(* Monitoring Prisma *)
	IF (T_Visu.T_PlcParam.dwActualPage = 430) THEN
		FailingEdgePrisma(CLK:=TRUE);
		RisingEdgePrisma(CLK:=(T_Visu.T_PlcParam.dwActualPage = 430));
		IF RisingEdgePrisma.Q THEN
		(* 0= 3 value prisma, 1 = 3 value prisma input para, 2 = 2 value prisma, 3 = 2 value prisma input para *)
			IF (T_Visu.ptrT_ExchgParam^.T_StationCommon.T_PrismPara.bStateInputPrisma = 1) THEN
				T_Visu.ptrT_ExchgParam^.T_StationCommon.T_PrismPara.bStateInputPrisma:=0;
			END_IF;
			IF (T_Visu.ptrT_ExchgParam^.T_StationCommon.T_PrismPara.bStateInputPrisma = 3) THEN
				T_Visu.ptrT_ExchgParam^.T_StationCommon.T_PrismPara.bStateInputPrisma:=2;
			END_IF;
		END_IF;
	ELSE
		RisingEdgePrisma(CLK:=FALSE);
		FailingEdgePrisma(CLK:=FALSE);
		(*If the page changes, then copy again the settled value *)
		IF FailingEdgePrisma.Q THEN
			T_Visu.ptrT_ExchgParam^.T_StationCommon.T_PrismPara:=T_NovRAM.T_Data.T_ProcessImageData.T_PrismPara;
		END_IF;
	END_IF

(* Tmp timer *)
	TimerONTmp(IN:=TRUE);



(************************************************************************************************************************************************************************)
(***************                                          start of the management for call a function of the visualisation interface                                           ********************)
(************************************************************************************************************************************************************************)
CtrlVisuFunction;
(************************************************************************************************************************************************************************)
(***************                                          end of the management for call a function of the visualisation interface                                           ********************)
(************************************************************************************************************************************************************************)



(************************************************************************************************************************************************************************)
(***************                                                   start of the checking of the activation of an visualisation action                                                   ********************)
(************************************************************************************************************************************************************************)
(* check if Action is Acitve and if the power supply is on, otherwise block the action *)
	xTmp:=	xStopAxis OR xMoveRelPosition OR xMoveAbsPosition OR xMoveContinousVel OR xSwitchMasterSlave OR xToggleAxisPower OR xResetAxis OR xReferenceAxis OR xTeachPosition OR xCylBrake;
	xTmp:=	xTmp OR xToggleCylinderState OR xToolTensForceAdd OR xToolTensForceAddMore OR xToolTensForceSub OR xToolTensForceSubMore;
	xTmp:=	xTmp OR xToolFeederMoveStartPos OR xToggleAllAxisPower OR xCalcAngleRefIndex OR xToolFeederMoveLoadPos;
	xTmp:=	xTmp OR xActivateStationFunction OR xActionProcStation OR xActionProcMachine OR xStopProcess;
	xTmp:=	xTmp OR xOverlayGrindFeedSetPlung OR xOverlayMeasureToolDia OR xFctCorrectionToolDiameter OR xAction_LoadProfileToProcessImage;
	xTmp:=	xTmp OR ((T_Visu.T_PlcParam.dwActualPage = 430) AND xAction_SaveNovRAM);
(*SOA 31.01.2023  { *)
	xTmp:= xTmp OR (T_Visu.T_PlcParam.dwActualPage = 141) ;
(*SOA 31.01.2023  } *)
	IF xTmp THEN
		IF NOT(T_TwinSafeOut.QxContactor_K3) OR NOT(T_TwinSafeOut.QxContactor_K4) THEN
			xStopAxis:=xMoveRelPosition:=xMoveAbsPosition:=xMoveContinousVel:=xSwitchMasterSlave:=xToggleAxisPower:=xResetAxis:=xReferenceAxis:=xTeachPosition:=xCylBrake:=FALSE;
			xToggleCylinderState:=xToolTensForceAdd:=xToolTensForceAddMore:=xToolTensForceSub:=xToolTensForceSubMore:=FALSE;
			xToolFeederMoveStartPos:=xToggleAllAxisPower:=xCalcAngleRefIndex:=xToolFeederMoveLoadPos:= FALSE;
			xActivateStationFunction:=xActionProcStation:=xActionProcMachine:=xStopProcess:=FALSE;
			xOverlayGrindFeedSetPlung:=xOverlayMeasureToolDia:=xFctCorrectionToolDiameter:=xAction_LoadProfileToProcessImage:=FALSE;
			T_Visu.ptrT_ExchgParam^.T_FunctionCommon.xOpenOverlayMessageBox:=FALSE;
			T_Visu.ptrT_ExchgParam^.T_FunctionCommon.xOpenOverlayMeasureInput:=FALSE;
			T_Visu.ptrT_ExchgParam^.T_FunctionCommon.xOpenOverlaySetGrindPlunge:=FALSE;
			T_Visu.ptrT_ExchgParam^.T_FunctionCommon.xSaveButton:=FALSE;
			T_Visu.ptrT_ExchgParam^.T_FunctionCommon.xExitButton:=FALSE;
			T_Visu.ptrT_ExchgParam^.T_FunctionCommon.xHideProgressbar:=FALSE;
			xAction_SaveNovRAM:=FALSE;
			T_Visu.T_CtrleAction.xDone:=TRUE;
			T_Visu.T_CtrleAction.xNotReady:=FALSE;
			T_Visu.T_CtrleAction.xErr:=FALSE;
			T_Visu.T_CtrleAction.udiErrorID:=0;
			tTimeOutAction:=T#0s;
			TimerAction(IN:=FALSE);
			(* Display Message --> Switch first the energy supply ON *)
			T_ExchgParam.T_Visu.T_Message.iState:=120;
			xBlockConfirmMessage:=TRUE;
			TONTimeWaitMsg(IN:=FALSE);
		END_IF;
	END_IF;
	IF (T_ExchgParam.T_Visu.T_Message.iState = 120) THEN
		TONTimeWaitMsg(IN:=TRUE,PT:=T#3s);
		IF TONTimeWaitMsg.Q THEN
			T_ExchgParam.T_Visu.T_Message.iState:=0;	(* Deactivate again the message *)
		END_IF;
	ELSE
		TONTimeWaitMsg(IN:=FALSE);
	END_IF;

(* check if an error is active, otherwise block the action *)
	IF (T_ExchgParam.T_Visu.T_Message.iState = 401) THEN
		xTmp:=	xStopAxis OR xMoveRelPosition OR xMoveAbsPosition OR xMoveContinousVel OR xSwitchMasterSlave OR xToggleAxisPower OR xResetAxis OR xReferenceAxis OR xTeachPosition OR xCylBrake;
		xTmp:=	xTmp OR xToggleCylinderState OR xToolTensForceAdd OR xToolTensForceAddMore OR xToolTensForceSub OR xToolTensForceSubMore;
		xTmp:=	xTmp OR xToolFeederMoveStartPos OR xToggleAllAxisPower OR xCalcAngleRefIndex OR xToolFeederMoveLoadPos;
		xTmp:=	xTmp OR xActivateStationFunction OR xActionProcStation OR xActionProcMachine OR xStopProcess;
		xTmp:=	xTmp OR xOverlayGrindFeedSetPlung OR xOverlayMeasureToolDia OR xFctCorrectionToolDiameter OR xAction_LoadProfileToProcessImage;
		xTmp:=	xTmp OR ((T_Visu.T_PlcParam.dwActualPage = 430) AND xAction_SaveNovRAM);
		IF xTmp THEN
			xStopAxis:=xMoveRelPosition:=xMoveAbsPosition:=xMoveContinousVel:=xSwitchMasterSlave:=xToggleAxisPower:=xResetAxis:=xReferenceAxis:=xTeachPosition:=xCylBrake:=FALSE;
			xToggleCylinderState:=xToolTensForceAdd:=xToolTensForceAddMore:=xToolTensForceSub:=xToolTensForceSubMore:=FALSE;
			xToolFeederMoveStartPos:=xToggleAllAxisPower:=xCalcAngleRefIndex:=xToolFeederMoveLoadPos:=FALSE;
			xActivateStationFunction:=xActionProcStation:=xActionProcMachine:=xStopProcess:=FALSE;
			xOverlayGrindFeedSetPlung:=xOverlayMeasureToolDia:=xFctCorrectionToolDiameter:=xAction_LoadProfileToProcessImage:=FALSE;
			xAction_SaveNovRAM:=FALSE;
			T_Visu.T_CtrleAction.xDone:=TRUE;
			T_Visu.T_CtrleAction.xNotReady:=FALSE;
			T_Visu.T_CtrleAction.xErr:=FALSE;
			T_Visu.T_CtrleAction.udiErrorID:=0;
			tTimeOutAction:=T#0s;
			TimerAction(IN:=FALSE);
		END_IF;
	END_IF;
(************************************************************************************************************************************************************************)
(***************                                                   end of the checking of the activation of an visualisation action                                                   ********************)
(************************************************************************************************************************************************************************)

(************************************************************************************************************************************************************************)
(***************                                             start for the section for defined function of the visualisation interface                                               ********************)
(************************************************************************************************************************************************************************)
VisuFunction_SetParameterPage;

(* Action change page from navigation panel *)
	IF xNavPanelChangePage OR xBtPanelLeftChangePage OR  xBtPanelRightChangePage OR xNextPageVertical THEN
		(* Step change page from navigation panel *)
		CASE iStepAction OF
		(* check visu *)
		1:	xTmp:=	T_Visu.T_CtrleVisu.xDone
					AND NOT(T_Visu.T_CtrleVisu.xExecute)
					AND NOT(T_Visu.T_CtrleVisu.xErr);
			IF xTmp THEN
				(* next Step *)
				iStepAction :=10;
				xStepActionDone:=FALSE;
			(* activ error *)
			ELSE iStepAction:=95; END_IF
		(* activ change page *)
		10:	T_Visu.T_CtrleVisu.xExecute:=TRUE;
			T_Visu.T_CtrleVisu.iFunction:=1;
			T_Visu.ptrT_ExchgParam^.T_Config.iEditParam:=0;
			IF xNavPanelChangePage THEN
				T_Visu.T_PlcParam.dwSetNewPage:=INT_TO_DWORD(T_Visu.T_CtrleAction.iFunction - 10000);
				CASE T_Visu.ptrT_ExchgParam^.T_Visu.bActivSpecialLayer OF
					0:	IF awNormalLayerActivPage[wTmpNormalLayerActivTask] <> 0 AND awNormalLayerActivPage[wTmpNormalLayerActivTask] <> T_Visu.T_PlcParam.dwSetNewPage THEN
							T_Visu.T_PlcParam.dwSetNewPage:=awNormalLayerActivPage[wTmpNormalLayerActivTask];
						END_IF;
					1:	IF awSpecialLayerGeneralActivPage[wTmpSpecialLayerGeneralActivTask] <> 0 AND awSpecialLayerGeneralActivPage[wTmpSpecialLayerGeneralActivTask] <> T_Visu.T_PlcParam.dwSetNewPage THEN
							T_Visu.T_PlcParam.dwSetNewPage:=awSpecialLayerGeneralActivPage[wTmpSpecialLayerGeneralActivTask];
						END_IF;
					2:	IF awSpecialLayerToolRotActivPage[wTmpSpecialLayerToolRotActivTask] <> 0 AND awSpecialLayerToolRotActivPage[wTmpSpecialLayerToolRotActivTask] <> T_Visu.T_PlcParam.dwSetNewPage THEN
							T_Visu.T_PlcParam.dwSetNewPage:=awSpecialLayerToolRotActivPage[wTmpSpecialLayerToolRotActivTask];
						END_IF;
					3:	IF awSpecialLayerWireFeedActivPage[wTmpSpecialLayerWireFeedActivTask] <> 0 AND awSpecialLayerWireFeedActivPage[wTmpSpecialLayerWireFeedActivTask] <> T_Visu.T_PlcParam.dwSetNewPage THEN
							T_Visu.T_PlcParam.dwSetNewPage:=awSpecialLayerWireFeedActivPage[wTmpSpecialLayerWireFeedActivTask];
						END_IF;
					4:	IF awSpecialLayerGrindAxisActivPage[wTmpSpecialLayerGrindAxisActivTask] <> 0 AND awSpecialLayerGrindAxisActivPage[wTmpSpecialLayerGrindAxisActivTask] <> T_Visu.T_PlcParam.dwSetNewPage THEN
							T_Visu.T_PlcParam.dwSetNewPage:=awSpecialLayerGrindAxisActivPage[wTmpSpecialLayerGrindAxisActivTask];
						END_IF;
				END_CASE;
			END_IF;
			IF xBtPanelLeftChangePage THEN
				T_Visu.T_PlcParam.dwSetNewPage:=dwSetNewPage;
				T_Visu.ptrT_ExchgParam^.T_Config.xBlockParaListNavi:=FALSE;
				T_Visu.ptrT_ExchgParam^.T_Config.xBlockParaListNavi1:=TRUE;
				T_Visu.ptrT_ExchgParam^.T_Config.xBlockProfilList:=TRUE;
			END_IF;
(*SOA*)
			IF xBtPanelRightChangePage THEN
				T_Visu.T_PlcParam.dwSetNewPage:=dwSetNewPage;
				T_Visu.ptrT_ExchgParam^.T_Config.xBlockParaListNavi:=FALSE;
				T_Visu.ptrT_ExchgParam^.T_Config.xBlockParaListNavi1:=TRUE;
				T_Visu.ptrT_ExchgParam^.T_Config.xBlockProfilList:=TRUE;
			END_IF;
(*SOA*)
			IF xNextPageVertical THEN
				IF (T_Visu.T_PageIndex[T_Visu.T_PlcParam.dwActualPage + 1].iIndexConfigPage <> 0) THEN
					T_Visu.T_PlcParam.dwSetNewPage:=T_Visu.T_PlcParam.dwActualPage + 1;
				ELSE
					FOR ii:=1 TO 9 DO
						IF (T_Visu.T_PageIndex[T_Visu.T_PlcParam.dwActualPage - 1].iIndexConfigPage <> 0) THEN
							T_Visu.T_PlcParam.dwActualPage:=T_Visu.T_PlcParam.dwActualPage - 1;
						ELSE
							T_Visu.T_PlcParam.dwSetNewPage:=T_Visu.T_PlcParam.dwActualPage;
							EXIT;
						END_IF;
					END_FOR;
				END_IF;
				CASE T_Visu.ptrT_ExchgParam^.T_Visu.bActivSpecialLayer OF
					0:	awNormalLayerActivPage[wTmpNormalLayerActivTask]:=DWORD_TO_WORD(T_Visu.T_PlcParam.dwSetNewPage);
					1:	awSpecialLayerGeneralActivPage[wTmpSpecialLayerGeneralActivTask]:=DWORD_TO_WORD(T_Visu.T_PlcParam.dwSetNewPage);
					2:	awSpecialLayerToolRotActivPage[wTmpSpecialLayerToolRotActivTask]:=DWORD_TO_WORD(T_Visu.T_PlcParam.dwSetNewPage);
					3:	awSpecialLayerWireFeedActivPage[wTmpSpecialLayerWireFeedActivTask]:=DWORD_TO_WORD(T_Visu.T_PlcParam.dwSetNewPage);
					4:	awSpecialLayerGrindAxisActivPage[wTmpSpecialLayerGrindAxisActivTask]:=DWORD_TO_WORD(T_Visu.T_PlcParam.dwSetNewPage);
				END_CASE;
			END_IF;
			(* next Step *)
			iStepAction :=20;
			xStepActionDone:=FALSE;
		(* wait  confirmation *)
		20:	IF NOT(xStepActionDone) THEN
				T_Visu.T_CtrleVisu.xExecute:=FALSE;
				(* confirm Step *)
				xStepActionDone:=TRUE;
			ELSE
				IF T_Visu.T_CtrleVisu.xDone THEN
				(* next Step *)
					iStepAction :=90;
					xStepActionDone:=FALSE;
				ELSE	IF T_Visu.T_CtrleVisu.xErr THEN
							iStepAction:=99;
							xStepActionDone:=FALSE;
						END_IF
				END_IF
			END_IF
		(* change page done *)
		90:	T_Visu.T_CtrleAction.xDone:=TRUE;
			T_Visu.T_CtrleAction.xNotReady:=FALSE;
			T_Visu.T_CtrleAction.xErr:=FALSE;
			T_Visu.T_CtrleAction.udiErrorID:=0;
			xNavPanelChangePage:=FALSE;
			xBtPanelLeftChangePage:=FALSE;
			xBtPanelRightChangePage:=FALSE;
			xNextPageVertical:=FALSE;
		(* visu not ready *)
		95:	T_Visu.T_CtrleAction.xDone:=TRUE;
			T_Visu.T_CtrleAction.xNotReady:=FALSE;
			T_Visu.T_CtrleAction.xErr:=FALSE;
			T_Visu.T_CtrleAction.udiErrorID:=0;
			xNavPanelChangePage:=FALSE;
			xBtPanelLeftChangePage:=FALSE;
			xBtPanelRightChangePage:=FALSE;
			xNextPageVertical:=FALSE;
		(* error *)
		99:	T_Visu.T_CtrleAction.xDone:=FALSE;
			T_Visu.T_CtrleAction.xNotReady:=FALSE;
			T_Visu.T_CtrleAction.xErr:=TRUE;
			T_Visu.T_CtrleAction.udiErrorID:=16#F0000 + T_Visu.T_CtrleAction.iFunction;
			xNavPanelChangePage:=FALSE;
			xBtPanelLeftChangePage:=FALSE;
			xBtPanelRightChangePage:=FALSE;
			xNextPageVertical:=FALSE;
		END_CASE
	END_IF

(* Action reset error station *)
	IF xResetError THEN
		(* FB clear error station *)
		fbQvisClearError(	xExecute:=xResetError,
						iError:=T_Visu.T_CtrleAction.iFunction,
						T_Message:=T_ExchgParam.T_Visu.T_Message,
						T_Station:=T_Station,
						T_Process:=T_Process,
						T_NovRAM:=T_NovRAM,
						T_Profile:=T_Profile,
						T_HDD:=T_HDD,
						xDone=>T_Visu.T_CtrleAction.xDone,
						xNotReady=>T_Visu.T_CtrleAction.xNotReady,
						xErr=>T_Visu.T_CtrleAction.xErr,
						udiErrorID=>T_Visu.T_CtrleAction.udiErrorID);
		IF T_Visu.T_CtrleAction.xDone OR T_Visu.T_CtrleAction.xNotReady OR T_Visu.T_CtrleAction.xErr THEN
			xResetError:=FALSE;
			fbQvisClearError(	xExecute:=xResetError,
							iError:=T_Visu.T_CtrleAction.iFunction,
							T_Message:=T_ExchgParam.T_Visu.T_Message,
							T_Station:=T_Station,
							T_Process:=T_Process,
							T_NovRAM:=T_NovRAM,
							T_Profile:=T_Profile,
							T_HDD:=T_HDD);
		END_IF
	END_IF

(* Action Delete Errorlist for Machine and Station *)
	IF xDeleteErrorList THEN
		(* Step saving NovRAM *)
		CASE iStepAction OF
		(* check NovRAM *)
		1:	xTmp:=	T_NovRAM.T_Ctrle.xDone
					AND NOT(T_NovRAM.T_Ctrle.xExecute)
					AND NOT(T_NovRAM.T_Ctrle.xErr);
			IF xTmp THEN
				(* next Step *)
				iStepAction :=10;
			(* activ error *)
			ELSE iStepAction:=95; END_IF
		10:	(* For delete the error, it need the system level *)
			IF (T_ExchgParam.T_Visu.T_Level.iActLevel <> 2) THEN
				T_ExchgParam.T_Visu.T_Message.iState:=42;	(* Display Message --> The error list may delete only in system level ! *)
				iStepAction:=90;
				RETURN;
			END_IF;
			T_Visu.ptrT_ExchgParam^.T_Visu.T_Message.iState:=108;	(* Confirm saving action <Enter>, or escape <Esc> ? *)
			(* next Step *)
			iStepAction :=20;
		(* waiting for saving confirmation key <Enter> or <Esc> *)
		20:	IF RisingEdgeKeyPanel_Enter.Q THEN
			(* Display message *)
				T_Visu.ptrT_ExchgParam^.T_Visu.T_Message.iState:=13;	(* Start saving *)
				(* next step *)
				iStepAction:=30;
			ELSE
				IF RisingEdgeKeyPanel_Esc.Q THEN iStepAction:=90; END_IF
				(* An other message has been displayed, stop saving action *)
				IF T_Visu.ptrT_ExchgParam^.T_Visu.T_Message.iState<>108 THEN iStepAction:=90; END_IF
			END_IF
		30:	FOR ii:=1 TO 20 DO
				T_NovRAM.T_Data.T_ErrorNrList.adiErrorListMachine[ii]:=0;
				T_NovRAM.T_Data.T_ErrorNrList.asErrorTimeStampMachine[ii]:='';
			END_FOR;
			(* activ save *)
			T_NovRAM.T_Ctrle.xExecute:=TRUE;
			T_NovRAM.T_Ctrle.iFunction:=2;
			(* next Step *)
			iStepAction :=40;
			xStepActionDone:=FALSE;
		(* wait save confirmation *)
		40:	IF NOT(xStepActionDone) THEN
				T_NovRAM.T_Ctrle.xExecute:=FALSE;
				(* confirm Step *)
				xStepActionDone:=TRUE;
			ELSE
				IF T_NovRAM.T_Ctrle.xDone THEN
				(* next Step *)
					iStepAction :=90;
					xStepActionDone:=FALSE;
					xUpdateErrorList:=TRUE;
				ELSE	IF T_NovRAM.T_Ctrle.xErr THEN
							iStepAction:=99;
							xStepActionDone:=FALSE;
						END_IF
				END_IF
			END_IF
		(* no code, waiting timeout *)
		89:	IF TimerAction.Q THEN iStepAction:=90; END_IF
		(* save done *)
		90:	IF (T_ExchgParam.T_Visu.T_Message.iState <> 42) THEN
				T_Visu.ptrT_ExchgParam^.T_Visu.T_Message.iState:=0;
			END_IF;
			T_Visu.T_CtrleAction.xDone:=TRUE;
			T_Visu.T_CtrleAction.xNotReady:=FALSE;
			T_Visu.T_CtrleAction.xErr:=FALSE;
			T_Visu.T_CtrleAction.udiErrorID:=0;
			xDeleteErrorList:=FALSE;
		(* NovRAM not ready *)
		95:	TimerNotReady(IN:=TRUE);
			xDeleteErrorList:=FALSE;
		(* error *)
		99:	T_Visu.T_CtrleAction.xDone:=FALSE;
			T_Visu.T_CtrleAction.xNotReady:=FALSE;
			T_Visu.T_CtrleAction.xErr:=TRUE;
			T_Visu.T_CtrleAction.udiErrorID:=16#F0000 + T_Visu.T_CtrleAction.iFunction;
			xDeleteErrorList:=FALSE;
		END_CASE;
	END_IF;

(* Open Overlay for input measured tool diameter *)
	IF xOverlayMeasureToolDia THEN
		CASE iStepAction OF
		(* check axis *)
		1:	IF NOT T_Station.TControl.xHardwareConfigError THEN
				xStepActionDone:=FALSE;
				iStepAction:=95;
				xTmp:=	T_Station.THardware.TAxisGrindFeeder.T_CtrleSingle.xDone
						AND T_Station.THardware.TAxisGrindFeeder.T_CtrleSingle.xReady
						AND T_Station.THardware.TAxisGrindFeeder.T_CtrleSingle.xNotMoving
						AND NOT(T_Station.THardware.TAxisGrindFeeder.T_CtrleSingle.xErr)
						AND NOT(T_Station.THardware.TAxisGrindFeeder.T_CtrleSingle.xExecute);
				(* Start/Stop position or speed of teachin page has to be confirmed *)
				IF xTmp THEN
					iStepAction:=10;
				END_IF
			ELSE
				iStepAction:=95;
			END_IF;
		10:	(* Open Overlay *)
			T_Visu.ptrT_ExchgParam^.T_FunctionCommon.xOpenOverlayMeasureInput:=TRUE;
			T_Visu.ptrT_ExchgParam^.T_FunctionCommon.xHideProgressbar:=TRUE;
			T_Visu.ptrT_ExchgParam^.T_FunctionCommon.rInputMeasToolDiameter:=T_Visu.ptrT_ExchgParam^.T_InfoValueCommon.rToolDiameter;
			(* next Step *)
			iStepAction :=20;
		20:	IF T_Visu.ptrT_ExchgParam^.T_FunctionCommon.xSaveButton THEN
				T_Visu.ptrT_ExchgParam^.T_FunctionCommon.xSaveButton:=FALSE;
				T_Visu.ptrT_ExchgParam^.T_FunctionCommon.xExitButton:=FALSE;
				(* next Step *)
				iStepAction :=30;
			END_IF;
			IF T_Visu.ptrT_ExchgParam^.T_FunctionCommon.xExitButton THEN
				T_Visu.ptrT_ExchgParam^.T_FunctionCommon.xSaveButton:=FALSE;
				T_Visu.ptrT_ExchgParam^.T_FunctionCommon.xExitButton:=FALSE;
				(* next Step *)
				iStepAction :=90;
			END_IF;
			IF T_Visu.T_CtrleAction.xDone THEN
				T_Visu.ptrT_ExchgParam^.T_FunctionCommon.xOpenOverlayMeasureInput:=FALSE;
				T_Visu.ptrT_ExchgParam^.T_FunctionCommon.xSaveButton:=FALSE;
				T_Visu.ptrT_ExchgParam^.T_FunctionCommon.xExitButton:=FALSE;
				T_Visu.ptrT_ExchgParam^.T_FunctionCommon.xHideProgressbar:=FALSE;
				xOverlayMeasureToolDia:=FALSE;
			END_IF;
		(* activ function axis *)
		30:	T_Station.THardware.TAxisGrindFeeder.T_CtrleSingle.rSetPosition:=	T_Station.THardware.TAxisGrindFeeder.T_LiveValue.lrActualPosition +
																		(T_Visu.ptrT_ExchgParam^.T_FunctionCommon.rInputMeasToolDiameter -
																		T_Visu.ptrT_ExchgParam^.T_InfoValueCommon.rToolDiameter);
			IF (T_Station.THardware.TAxisGrindFeeder.T_CtrleSingle.rSetPosition < T_NovRAM.T_Data.T_ProcessImageData.T_PrismPara.rToolDiameterMin) OR
			     (T_Station.THardware.TAxisGrindFeeder.T_CtrleSingle.rSetPosition > (T_NovRAM.T_Data.T_ProcessImageData.T_PrismPara.rToolDiameterMax + T_NovRAM.T_Data.T_Standard.T_TeachINGrindFeeder.rOffsetSWPosEndSwitch)) THEN
				T_Visu.ptrT_ExchgParam^.T_Visu.T_Message.iState:=123;	(* Out of Range, GrindFeeder position not settled! *)
				iStepAction:=50;
			ELSE
				T_Station.THardware.TAxisGrindFeeder.T_CtrleSingle.iFunction:=11;
				T_Station.THardware.TAxisGrindFeeder.T_CtrleSingle.xExecute:=TRUE;
				(* next step *)
				iStepAction:=50;
			END_IF;
			xStepActionDone:=FALSE;
		(* confirm execution *)
		50:	IF NOT(xStepActionDone) THEN
			(* confirm execution *)
				T_Station.THardware.TAxisGrindFeeder.T_CtrleSingle.xExecute:=FALSE;
				xStepActionDone:=TRUE;
			ELSE
				IF T_Station.THardware.TAxisGrindFeeder.T_CtrleSingle.xDone THEN
				(* confirm action next step *)
					iStepAction:=90;
					xStepActionDone:=FALSE;
				ELSE
					IF T_Station.THardware.TAxisGrindFeeder.T_CtrleSingle.xErr THEN
					(* activ action not ready or error *)
						iStepAction:=99;
						xStepActionDone:=FALSE;
					END_IF
				END_IF
			END_IF
		(* action done *)
		90:	T_Visu.ptrT_ExchgParam^.T_StationCommon.wState:=T_Visu.ptrT_ExchgParam^.T_StationCommon.wState AND 16#BF;
			T_Visu.T_CtrleAction.xDone:=TRUE;
			T_Visu.T_CtrleAction.xNotReady:=FALSE;
			T_Visu.T_CtrleAction.xErr:=FALSE;
			T_Visu.T_CtrleAction.udiErrorID:=0;
			xOverlayMeasureToolDia:=FALSE;
			T_Visu.ptrT_ExchgParam^.T_FunctionCommon.xOpenOverlayMeasureInput:=FALSE;
			T_Visu.ptrT_ExchgParam^.T_FunctionCommon.xHideProgressbar:=FALSE;
		(* axis not ready *)
		95:	T_Visu.ptrT_ExchgParam^.T_StationCommon.wState:=T_Visu.ptrT_ExchgParam^.T_StationCommon.wState AND 16#BF;
			TimerNotReady(IN:=TRUE);
			xOverlayMeasureToolDia:=FALSE;
			T_Visu.ptrT_ExchgParam^.T_FunctionCommon.xOpenOverlayMeasureInput:=FALSE;
			T_Visu.ptrT_ExchgParam^.T_FunctionCommon.xHideProgressbar:=FALSE;
		(* error *)
		99:	T_Visu.ptrT_ExchgParam^.T_StationCommon.wState:=T_Visu.ptrT_ExchgParam^.T_StationCommon.wState AND 16#BF;
			T_Visu.T_CtrleAction.xDone:=TRUE;
			T_Visu.T_CtrleAction.xNotReady:=FALSE;
			IF (T_Station.THardware.TAxisGrindFeeder.T_Config_Gen.iTyp <> 0) THEN
				diErrorNr:=(T_Station.THardware.TAxisGrindFeeder.T_Config_Gen.iTyp * 1000000) + T_Station.THardware.TAxisGrindFeeder.T_CtrleSingle.udiErrorID;
			ELSE
				diErrorNr:=0;
			END_IF;
			FBErrorMessage(	diErrorNr:=diErrorNr,
							T_ErrorList:=T_ErrorList);
			T_Visu.ptrT_ExchgParam^.T_Visu.T_Message.sDynamicTextEnglish:=FBErrorMessage.sErrorTextEnglish;
			T_Visu.ptrT_ExchgParam^.T_Visu.T_Message.sDynamicTextDeutsch:=FBErrorMessage.sErrorTextDeutsch;
			T_Visu.ptrT_ExchgParam^.T_Visu.T_Message.sDynamicTextFrancais:=FBErrorMessage.sErrorTextFrancais;
			T_Visu.ptrT_ExchgParam^.T_SafetyCtrl.xSetForceError:=TRUE;
			T_Visu.ptrT_ExchgParam^.T_SafetyCtrl.diSetForceErrorNr:=diErrorNr;
			T_Visu.T_CtrleAction.xErr:=FALSE;
			T_Visu.T_CtrleAction.udiErrorID:=0;
			T_Station.THardware.TAxisGrindFeeder.T_CtrleSingle.iFunction:=1;
			T_Station.THardware.TAxisGrindFeeder.T_CtrleSingle.xExecute:=TRUE;
			xOverlayMeasureToolDia:=FALSE;
			T_Visu.ptrT_ExchgParam^.T_FunctionCommon.xOpenOverlayMeasureInput:=FALSE;
			T_Visu.ptrT_ExchgParam^.T_FunctionCommon.xHideProgressbar:=FALSE;
		END_CASE
	END_IF;

(* Open Overlay for input the correction of the position of the GrindFeeder *)
	IF xOverlayGrindFeedSetPlung THEN
		CASE iStepAction OF
		(* check axis *)
		1:	IF NOT T_Station.TControl.xHardwareConfigError THEN
				xStepActionDone:=FALSE;
				iStepAction:=95;
				xTmp:=	T_Station.THardware.TAxisGrindFeeder.T_CtrleSingle.xDone
						AND T_Station.THardware.TAxisGrindFeeder.T_CtrleSingle.xReady
						AND T_Station.THardware.TAxisGrindFeeder.T_CtrleSingle.xNotMoving
						AND NOT(T_Station.THardware.TAxisGrindFeeder.T_CtrleSingle.xErr)
						AND NOT(T_Station.THardware.TAxisGrindFeeder.T_CtrleSingle.xExecute);
				(* Start/Stop position or speed of teachin page has to be confirmed *)
				IF xTmp THEN
					iStepAction:=10;
				END_IF
			ELSE
				iStepAction:=95;
			END_IF;
		10:	(* Open Overlay *)
			T_Visu.ptrT_ExchgParam^.T_FunctionCommon.xOpenOverlaySetGrindPlunge:=TRUE;
			T_Visu.ptrT_ExchgParam^.T_FunctionCommon.xHideProgressbar:=TRUE;
			T_Visu.ptrT_ExchgParam^.T_FunctionCommon.rInputGrindPlunge:=T_NovRAM.T_Data.T_ProcessImageData.T_CalibrationPara.rPlungeLengthGrindFeedCalib;
			(* next Step *)
			iStepAction :=20;
		20:	IF T_Visu.ptrT_ExchgParam^.T_FunctionCommon.xSaveButton THEN
				T_Visu.ptrT_ExchgParam^.T_FunctionCommon.xSaveButton:=FALSE;
				T_Visu.ptrT_ExchgParam^.T_FunctionCommon.xExitButton:=FALSE;
				(* next Step *)
				iStepAction :=30;
			END_IF;
			IF T_Visu.ptrT_ExchgParam^.T_FunctionCommon.xExitButton THEN
				T_Visu.ptrT_ExchgParam^.T_FunctionCommon.xSaveButton:=FALSE;
				T_Visu.ptrT_ExchgParam^.T_FunctionCommon.xExitButton:=FALSE;
				(* next Step *)
				iStepAction :=90;
			END_IF;
			IF T_Visu.T_CtrleAction.xDone THEN
				T_Visu.ptrT_ExchgParam^.T_FunctionCommon.xOpenOverlaySetGrindPlunge:=FALSE;
				T_Visu.ptrT_ExchgParam^.T_FunctionCommon.xSaveButton:=FALSE;
				T_Visu.ptrT_ExchgParam^.T_FunctionCommon.xExitButton:=FALSE;
				T_Visu.ptrT_ExchgParam^.T_FunctionCommon.xHideProgressbar:=FALSE;
				xOverlayGrindFeedSetPlung:=FALSE;
			END_IF;
		(* activ function axis *)
		30:	T_Station.THardware.TAxisGrindFeeder.T_CtrleSingle.rSetPosition:=	T_Station.THardware.TAxisGrindFeeder.T_LiveValue.lrActualPosition +
																		T_Visu.ptrT_ExchgParam^.T_FunctionCommon.rInputGrindPlunge;
			T_Station.THardware.TAxisGrindFeeder.T_CtrleSingle.iFunction:=11;
			T_Station.THardware.TAxisGrindFeeder.T_CtrleSingle.xExecute:=TRUE;
			(* next step *)
			iStepAction:=50;
			xStepActionDone:=FALSE;
		(* confirm execution *)
		50:	IF NOT(xStepActionDone) THEN
			(* confirm execution *)
				T_Station.THardware.TAxisGrindFeeder.T_CtrleSingle.xExecute:=FALSE;
				xStepActionDone:=TRUE;
			ELSE
				IF T_Station.THardware.TAxisGrindFeeder.T_CtrleSingle.xDone THEN
				(* confirm action next step *)
					iStepAction:=90;
					xStepActionDone:=FALSE;
				ELSE
					IF T_Station.THardware.TAxisGrindFeeder.T_CtrleSingle.xErr THEN
					(* activ action not ready or error *)
						iStepAction:=99;
						xStepActionDone:=FALSE;
					END_IF
				END_IF
			END_IF
		(* action done *)
		90:	T_Visu.ptrT_ExchgParam^.T_StationCommon.wState:=T_Visu.ptrT_ExchgParam^.T_StationCommon.wState AND 16#BF;
			T_Visu.T_CtrleAction.xDone:=TRUE;
			T_Visu.T_CtrleAction.xNotReady:=FALSE;
			T_Visu.T_CtrleAction.xErr:=FALSE;
			T_Visu.T_CtrleAction.udiErrorID:=0;
			xOverlayGrindFeedSetPlung:=FALSE;
			T_Visu.ptrT_ExchgParam^.T_FunctionCommon.xOpenOverlaySetGrindPlunge:=FALSE;
			T_Visu.ptrT_ExchgParam^.T_FunctionCommon.xHideProgressbar:=FALSE;
		(* axis not ready *)
		95:	T_Visu.ptrT_ExchgParam^.T_StationCommon.wState:=T_Visu.ptrT_ExchgParam^.T_StationCommon.wState AND 16#BF;
			TimerNotReady(IN:=TRUE);
			xOverlayGrindFeedSetPlung:=FALSE;
			T_Visu.ptrT_ExchgParam^.T_FunctionCommon.xOpenOverlaySetGrindPlunge:=FALSE;
			T_Visu.ptrT_ExchgParam^.T_FunctionCommon.xHideProgressbar:=FALSE;
		(* error *)
		99:	T_Visu.ptrT_ExchgParam^.T_StationCommon.wState:=T_Visu.ptrT_ExchgParam^.T_StationCommon.wState AND 16#BF;
			T_Visu.T_CtrleAction.xDone:=TRUE;
			T_Visu.T_CtrleAction.xNotReady:=FALSE;
			IF (T_Station.THardware.TAxisGrindFeeder.T_Config_Gen.iTyp <> 0) THEN
				diErrorNr:=(T_Station.THardware.TAxisGrindFeeder.T_Config_Gen.iTyp * 1000000) + T_Station.THardware.TAxisGrindFeeder.T_CtrleSingle.udiErrorID;
			ELSE
				diErrorNr:=0;
			END_IF;
			FBErrorMessage(	diErrorNr:=diErrorNr,
							T_ErrorList:=T_ErrorList);
			T_Visu.ptrT_ExchgParam^.T_Visu.T_Message.sDynamicTextEnglish:=FBErrorMessage.sErrorTextEnglish;
			T_Visu.ptrT_ExchgParam^.T_Visu.T_Message.sDynamicTextDeutsch:=FBErrorMessage.sErrorTextDeutsch;
			T_Visu.ptrT_ExchgParam^.T_Visu.T_Message.sDynamicTextFrancais:=FBErrorMessage.sErrorTextFrancais;
			T_Visu.ptrT_ExchgParam^.T_SafetyCtrl.xSetForceError:=TRUE;
			T_Visu.ptrT_ExchgParam^.T_SafetyCtrl.diSetForceErrorNr:=diErrorNr;
			T_Visu.T_CtrleAction.xErr:=FALSE;
			T_Visu.T_CtrleAction.udiErrorID:=0;
			T_Station.THardware.TAxisGrindFeeder.T_CtrleSingle.iFunction:=1;
			T_Station.THardware.TAxisGrindFeeder.T_CtrleSingle.xExecute:=TRUE;
			xOverlayGrindFeedSetPlung:=FALSE;
			T_Visu.ptrT_ExchgParam^.T_FunctionCommon.xOpenOverlaySetGrindPlunge:=FALSE;
			T_Visu.ptrT_ExchgParam^.T_FunctionCommon.xHideProgressbar:=FALSE;
		END_CASE
	END_IF;

(* Plunge On/Off or Displace On/Off *)
	IF xPlungeActivation OR xDisplaceActivation THEN
		CASE iStepAction OF
		(* check visu *)
		1:	xTmp:=	TRUE;
			IF xTmp THEN
				(* next Step *)
				iStepAction :=10;
			(* activ error *)
			ELSE iStepAction:=95; END_IF
		10:	(* Open Overlay *)
			IF xPlungeActivation THEN
				IF (T_Visu.T_PlcParam.dwActualPage = 110) THEN
					T_Visu.ptrT_ExchgParam^.T_StationCommon.T_CalibrationPara.xPlungeActivationCalib:=NOT(T_Visu.ptrT_ExchgParam^.T_StationCommon.T_CalibrationPara.xPlungeActivationCalib);
				ELSIF (T_Visu.T_PlcParam.dwActualPage = 10) THEN
					T_Visu.ptrT_ExchgParam^.T_StationCommon.T_AutoGeometryPara.xPlungeActivationGeometry:=NOT(T_Visu.ptrT_ExchgParam^.T_StationCommon.T_AutoGeometryPara.xPlungeActivationGeometry);
				ELSIF (T_Visu.T_PlcParam.dwActualPage = 20) THEN
					T_Visu.ptrT_ExchgParam^.T_StationCommon.T_AutoGroovePara.xPlungeActivationGroove:=NOT(T_Visu.ptrT_ExchgParam^.T_StationCommon.T_AutoGroovePara.xPlungeActivationGroove);
				END_IF;
			END_IF;
			IF xDisplaceActivation THEN
				IF (T_Visu.T_PlcParam.dwActualPage = 110) THEN
					T_Visu.ptrT_ExchgParam^.T_StationCommon.T_CalibrationPara.xDisplaceActivationCalib:=NOT(T_Visu.ptrT_ExchgParam^.T_StationCommon.T_CalibrationPara.xDisplaceActivationCalib);
				ELSIF (T_Visu.T_PlcParam.dwActualPage = 10) THEN
					T_Visu.ptrT_ExchgParam^.T_StationCommon.T_AutoGeometryPara.xDisplaceActivationGeometry:=NOT(T_Visu.ptrT_ExchgParam^.T_StationCommon.T_AutoGeometryPara.xDisplaceActivationGeometry);
				ELSIF (T_Visu.T_PlcParam.dwActualPage = 20) THEN
					T_Visu.ptrT_ExchgParam^.T_StationCommon.T_AutoGroovePara.xDisplaceActivationGroove:=NOT(T_Visu.ptrT_ExchgParam^.T_StationCommon.T_AutoGroovePara.xDisplaceActivationGroove);
				END_IF;
			END_IF;
			(* next Step *)
			iStepAction :=30;
		(* active saving data NovRAM *)
		30:	xAction_SaveNovRAM:=TRUE;
			iStepActionNovRam:=1;
			(* next step *)
			iStepAction:=40;
		(* waiting confirm saving NovRAM action *)
		40:	IF NOT xAction_SaveNovRAM THEN
				xCalcAgainProcTime:=TRUE;
				iStepAction:=90;
			END_IF;
		(* change page done *)
		90:	T_Visu.T_CtrleAction.xDone:=TRUE;
			T_Visu.T_CtrleAction.xNotReady:=FALSE;
			T_Visu.T_CtrleAction.xErr:=FALSE;
			T_Visu.T_CtrleAction.udiErrorID:=0;
			xPlungeActivation:=FALSE;
			xDisplaceActivation:=FALSE;
		(* not ready *)
		95:	T_Visu.T_CtrleAction.xDone:=TRUE;
			T_Visu.T_CtrleAction.xNotReady:=FALSE;
			T_Visu.T_CtrleAction.xErr:=FALSE;
			T_Visu.T_CtrleAction.udiErrorID:=0;
			xPlungeActivation:=FALSE;
			xDisplaceActivation:=FALSE;
		END_CASE
	END_IF;

(* AutoGroove-->Block GrindFeeder On/Off *)
	IF xBlockGrindFeederActivation THEN
		CASE iStepAction OF
		(* check visu *)
		1:	xTmp:=	TRUE;
			IF xTmp THEN
				(* next Step *)
				iStepAction :=10;
			(* activ error *)
			ELSE iStepAction:=95; END_IF
		10:	(* Open Overlay *)
			T_Visu.ptrT_ExchgParam^.T_StationCommon.T_AutoGroovePara.xBlockGrindFeeder:=NOT(T_Visu.ptrT_ExchgParam^.T_StationCommon.T_AutoGroovePara.xBlockGrindFeeder);
			(* next Step *)
			iStepAction :=30;
		(* active saving data NovRAM *)
		30:	xAction_SaveNovRAM:=TRUE;
			iStepActionNovRam:=1;
			(* next step *)
			iStepAction:=40;
		(* waiting confirm saving NovRAM action *)
		40:	IF NOT xAction_SaveNovRAM THEN
				iStepAction:=90;
			END_IF;
		(* change page done *)
		90:	T_Visu.T_CtrleAction.xDone:=TRUE;
			T_Visu.T_CtrleAction.xNotReady:=FALSE;
			T_Visu.T_CtrleAction.xErr:=FALSE;
			T_Visu.T_CtrleAction.udiErrorID:=0;
			xBlockGrindFeederActivation:=FALSE;
		(* not ready *)
		95:	T_Visu.T_CtrleAction.xDone:=TRUE;
			T_Visu.T_CtrleAction.xNotReady:=FALSE;
			T_Visu.T_CtrleAction.xErr:=FALSE;
			T_Visu.T_CtrleAction.udiErrorID:=0;
			xBlockGrindFeederActivation:=FALSE;
		END_CASE
	END_IF;

(* AutoGroove-->ToolFeeder move to StartPos *)
	IF xToolFeederMoveStartPos OR xToolFeederMoveLoadPos THEN
		(* Step move abs position *)
		CASE iStepAction OF
		(* check axis *)
		1:	IF NOT T_Station.TControl.xHardwareConfigError THEN
				xStepActionDone:=FALSE;
				iStepAction:=95;
				xTmp:=	T_Station.THardware.TAxisToolFeeder.T_CtrleSingle.xDone
						AND T_Station.THardware.TAxisToolFeeder.T_CtrleSingle.xReady
						AND T_Station.THardware.TAxisToolFeeder.T_CtrleSingle.xNotMoving
						AND T_Station.THardware.TAxisToolFeeder.T_CtrleSingle.xPower
						AND NOT(T_Station.THardware.TAxisToolFeeder.T_CtrleSingle.xErr)
						AND NOT(T_Station.THardware.TAxisToolFeeder.T_CtrleSingle.xExecute)
						AND ((T_Station.THardware.TAxisToolFeeder.T_CtrleSingle.xRef AND xMicroRodActive) OR NOT(xMicroRodActive));
				(* Start/Stop position or speed of teachin page has to be confirmed *)
				IF xTmp THEN
					iStepAction:=10;
				ELSE
					IF NOT T_Station.THardware.TAxisToolFeeder.T_CtrleSingle.xRef THEN
					(* Display message, axis not referenced *)
						tTimeOutAction:=TimerAction.ET+T#2s;
						T_Visu.ptrT_ExchgParam^.T_Visu.T_Message.iState:=18;
						(* Action has been cancelled *)
						iStepAction:=89;
					END_IF
				END_IF
			ELSE
				iStepAction:=95;
			END_IF;
		(* activ function axis *)
		10:	tTimeOutAction:=T#999s;
			bStateMachine:=2;
			xSetStateMachine:=TRUE;
			IF xMicroRodActive THEN
				iStepAction:=20;		(* Move Absolut *)
			END_IF;
			IF NOT(xMicroRodActive) THEN
				iStepAction:=35;		(* Move Relativ *)
			END_IF;
			(* init. acc/dec/jerk *)
			T_Station.THardware.TAxisToolFeeder.T_CtrleSingle.lrAcceleration:=T_NovRam.T_Data.T_Standard.T_TeachINToolFeeder.rAcceleration;
			T_Station.THardware.TAxisToolFeeder.T_CtrleSingle.lrDecceleration:=T_NovRam.T_Data.T_Standard.T_TeachINToolFeeder.rDeceleration;
			(*
			T_Station.THardware.TAxisToolFeeder.T_CtrleSingle.lrAcceleration:=T_Station.THardware.TAxisToolFeeder.T_Config_ObjFileValue.lrAcceleration;
			T_Station.THardware.TAxisToolFeeder.T_CtrleSingle.lrDecceleration:=T_Station.THardware.TAxisToolFeeder.T_Config_ObjFileValue.lrDecceleration;
			T_Station.THardware.TAxisToolFeeder.T_CtrleSingle.lrJerk:=T_Station.THardware.TAxisToolFeeder.T_Config_ObjFileValue.lrJerk;
			*)
		(* activ function axis move absolut *)
		20:	IF xToolFeederMoveStartPos THEN
				IF (T_Visu.T_PlcParam.dwActualPage = 10) THEN
					T_Station.THardware.TAxisToolFeeder.T_CtrleSingle.lrPosition:=	T_NovRam.T_Data.T_ProcessImageData.T_ProcessPara.rStartPosToolFeedAuto;
				END_IF;
				IF (T_Visu.T_PlcParam.dwActualPage = 20) THEN
					IF T_NovRam.T_Data.T_ProcessImageData.T_AutoGroovePara.xPlungeActivationGroove AND T_NovRam.T_Data.T_ProcessImageData.T_AutoGroovePara.xBlockGrindFeeder THEN
						T_Station.THardware.TAxisToolFeeder.T_CtrleSingle.lrPosition:=	T_NovRam.T_Data.T_ProcessImageData.T_ProcessPara.rStartPosToolFeedAuto +
																				T_NovRam.T_Data.T_ProcessImageData.T_AutoGroovePara.rPlungeLengthToolFeedGroove;
					ELSE
						T_Station.THardware.TAxisToolFeeder.T_CtrleSingle.lrPosition:=	T_NovRam.T_Data.T_ProcessImageData.T_ProcessPara.rStartPosToolFeedAuto;
					END_IF;
				END_IF;
				IF (T_Visu.T_PlcParam.dwActualPage = 110) THEN
					T_Station.THardware.TAxisToolFeeder.T_CtrleSingle.lrPosition:=	T_NovRam.T_Data.T_ProcessImageData.T_CalibrationPara.rStartPosToolFeedCalib;
				END_IF;
				T_Station.THardware.TAxisToolFeeder.T_CtrleSingle.lrVelocity:=T_NovRam.T_Data.T_ProcessImageData.T_ProcessPara.rSpeedStartPosToolFeedProcess;
			END_IF;
			IF xToolFeederMoveLoadPos THEN
				T_Station.THardware.TAxisToolFeeder.T_CtrleSingle.lrPosition:=	T_NovRam.T_Data.T_Standard.T_AxisPosition.rLoadPosToolFeedAuto;
				T_Station.THardware.TAxisToolFeeder.T_CtrleSingle.lrVelocity:=T_NovRam.T_Data.T_Standard.T_TeachINToolFeeder.rPositionSpeed;
			END_IF;
			T_Station.THardware.TAxisToolFeeder.T_CtrleSingle.iFunction:=7;
			T_Station.THardware.TAxisToolFeeder.T_CtrleSingle.xExecute:=TRUE;
			(* next step *)
			iStepAction:=40;
			xStepActionDone:=FALSE;
		(* activ function axis move relativ *)
		35:	IF (T_Visu.T_PlcParam.dwActualPage = 10) THEN
				T_Station.THardware.TAxisToolFeeder.T_CtrleSingle.lrDistance:=0;
			END_IF;
			IF (T_Visu.T_PlcParam.dwActualPage = 20) THEN
				IF T_NovRam.T_Data.T_ProcessImageData.T_AutoGroovePara.xPlungeActivationGroove (*AND T_NovRam.T_Data.T_ProcessImageData.T_AutoGroovePara.xBlockGrindFeeder*) THEN
					T_Station.THardware.TAxisToolFeeder.T_CtrleSingle.lrDistance:=T_NovRam.T_Data.T_ProcessImageData.T_AutoGroovePara.rPlungeLengthToolFeedGroove;
				ELSE
					(*T_Station.THardware.TAxisToolFeeder.T_CtrleSingle.lrDistance:=0;*)
					iStepAction:=95;
					RETURN;
				END_IF;
			END_IF;
			T_Station.THardware.TAxisToolFeeder.T_CtrleSingle.lrVelocity:=T_NovRam.T_Data.T_ProcessImageData.T_ProcessPara.rSpeedStartPosToolFeedProcess;
			T_Station.THardware.TAxisToolFeeder.T_CtrleSingle.iFunction:=8;
			T_Station.THardware.TAxisToolFeeder.T_CtrleSingle.xExecute:=TRUE;
			(* next step *)
			iStepAction:=40;
			xStepActionDone:=FALSE;
		(* confirm execution *)
		40:	IF NOT(xStepActionDone) THEN
			(* confirm execution *)
				T_Station.THardware.TAxisToolFeeder.T_CtrleSingle.xExecute:=FALSE;
				xStepActionDone:=TRUE;
				(* Display message, 'Start moving' *)
				T_Visu.ptrT_ExchgParam^.T_Visu.T_Message.iState:=26;
			ELSE
				IF T_Station.THardware.TAxisToolFeeder.T_CtrleSingle.xDone THEN
				(* confirm action next step *)
					bStateMachine:=1;
					xSetStateMachine:=TRUE;
					iStepAction:=90;
					xStepActionDone:=FALSE;
				ELSE
					IF T_Station.THardware.TAxisToolFeeder.T_CtrleSingle.xErr THEN
					(* activ action not ready or error *)
						iStepAction:=99;
						xStepActionDone:=FALSE;
					END_IF
				END_IF
			END_IF
		(* waiting timeout *)
		89: IF TimerAction.Q THEN iStepAction:=90; END_IF
			(*T_Visu.ptrT_ExchgParam^.T_TeachIn.iStateAxisMovement:=1;*)
		(* action done *)
		90:	T_Visu.ptrT_ExchgParam^.T_StationCommon.wState:=T_Visu.ptrT_ExchgParam^.T_StationCommon.wState AND 16#BF;
			T_Visu.T_CtrleAction.xDone:=TRUE;
			T_Visu.T_CtrleAction.xNotReady:=FALSE;
			T_Visu.T_CtrleAction.xErr:=FALSE;
			T_Visu.T_CtrleAction.udiErrorID:=0;
			xToolFeederMoveStartPos:=xToolFeederMoveLoadPos:=FALSE;
			(*T_Visu.ptrT_ExchgParam^.T_TeachIn.iStateAxisMovement:=1;*)
		(* axis not ready *)
		95:	T_Visu.ptrT_ExchgParam^.T_StationCommon.wState:=T_Visu.ptrT_ExchgParam^.T_StationCommon.wState AND 16#BF;
			TimerNotReady(IN:=TRUE);
			xToolFeederMoveStartPos:=xToolFeederMoveLoadPos:=FALSE;
			(*T_Visu.ptrT_ExchgParam^.T_TeachIn.iStateAxisMovement:=1;*)
		(* error *)
		99:	T_Visu.ptrT_ExchgParam^.T_StationCommon.wState:=T_Visu.ptrT_ExchgParam^.T_StationCommon.wState AND 16#BF;
			T_Visu.T_CtrleAction.xDone:=TRUE;
			T_Visu.T_CtrleAction.xNotReady:=FALSE;
			IF (T_Station.THardware.TAxisToolFeeder.T_Config_Gen.iTyp <> 0) THEN
				diErrorNr:=(T_Station.THardware.TAxisToolFeeder.T_Config_Gen.iTyp * 1000000) + T_Station.THardware.TAxisToolFeeder.T_CtrleSingle.udiErrorID;
			ELSE
				diErrorNr:=0;
			END_IF;
			FBErrorMessage(	diErrorNr:=diErrorNr,
							T_ErrorList:=T_ErrorList);
			T_Visu.ptrT_ExchgParam^.T_Visu.T_Message.sDynamicTextEnglish:=FBErrorMessage.sErrorTextEnglish;
			T_Visu.ptrT_ExchgParam^.T_Visu.T_Message.sDynamicTextDeutsch:=FBErrorMessage.sErrorTextDeutsch;
			T_Visu.ptrT_ExchgParam^.T_Visu.T_Message.sDynamicTextFrancais:=FBErrorMessage.sErrorTextFrancais;
			T_Visu.ptrT_ExchgParam^.T_SafetyCtrl.xSetForceError:=TRUE;
			T_Visu.ptrT_ExchgParam^.T_SafetyCtrl.diSetForceErrorNr:=diErrorNr;
			T_Visu.T_CtrleAction.xErr:=FALSE;
			T_Visu.T_CtrleAction.udiErrorID:=0;
			T_Station.THardware.TAxisToolFeeder.T_CtrleSingle.iFunction:=1;
			T_Station.THardware.TAxisToolFeeder.T_CtrleSingle.xExecute:=TRUE;
			xToolFeederMoveStartPos:=xToolFeederMoveLoadPos:=FALSE;
			(*T_Visu.ptrT_ExchgParam^.T_TeachIn.iStateAxisMovement:=1;*)
		END_CASE
	END_IF
(*08.07.2014: KFS	{	*)
(* WarmUp On/Off*)
	IF xWarmUp THEN
		CASE iStepAction OF
		(* check visu *)
		1:	xTmp:=	TRUE;
			IF xTmp THEN
				(* next Step *)
				iStepAction :=10;
			(* activ error *)
			ELSE iStepAction:=95; END_IF
		10:	(* Open Overlay *)
			IF (T_Visu.T_PlcParam.dwActualPage = 10) THEN
				T_Visu.ptrT_ExchgParam^.T_StationCommon.T_AutoGeometryPara.xWarmUp:=NOT(T_Visu.ptrT_ExchgParam^.T_StationCommon.T_AutoGeometryPara.xWarmUp);
			END_IF;
			(* next Step *)
			iStepAction :=90;
		(* change page done *)
		90:	T_Visu.T_CtrleAction.xDone:=TRUE;
			T_Visu.T_CtrleAction.xNotReady:=FALSE;
			T_Visu.T_CtrleAction.xErr:=FALSE;
			T_Visu.T_CtrleAction.udiErrorID:=0;
			xWarmUp:=FALSE;
		(* not ready *)
		95:	T_Visu.T_CtrleAction.xDone:=TRUE;
			T_Visu.T_CtrleAction.xNotReady:=FALSE;
			T_Visu.T_CtrleAction.xErr:=FALSE;
			T_Visu.T_CtrleAction.udiErrorID:=0;
			xWarmUp:=FALSE;
		END_CASE
	END_IF;
(*08.07.2014: KFS	}	*)

(*23.02.2023: SOA  {   Reset Warmup if Change of page   *)
IF (T_Visu.T_PlcParam.dwActualPage <> 10) THEN
	T_Visu.ptrT_ExchgParam^.T_StationCommon.T_AutoGeometryPara.xWarmUp := xWarmUp := xWarmUpMessage := xWarmUpMessageActiv := xWarmUpMessageDone := FALSE;
END_IF
(*23.02.2023: SOA  {      *)

(* AutoGeometry and AutoGroove-->Switch On/Off all Axis Power *)
	IF xToggleAllAxisPower THEN
		(* Step toggle Axis power *)
		CASE iStepAction OF
		(* check axis *)
		1:	IF NOT T_Station.TControl.xHardwareConfigError THEN
				xStepActionDone:=FALSE;
				iStepAction:=95;
				xTmp:=	T_Station.THardware.TAxisToolLeft.T_CtrleSingle.xDone
						AND T_Station.THardware.TAxisToolLeft.T_CtrleSingle.xNotMoving
						AND NOT(T_Station.THardware.TAxisToolLeft.T_CtrleSingle.xErr)
						AND NOT(T_Station.THardware.TAxisToolLeft.T_CtrleSingle.xExecute);
				xTmp:=	xTmp AND ((T_Station.THardware.TAxisToolCenter.T_CtrleSingle.xDone
						AND T_Station.THardware.TAxisToolCenter.T_CtrleSingle.xNotMoving
						AND NOT(T_Station.THardware.TAxisToolCenter.T_CtrleSingle.xErr)
						AND NOT(T_Station.THardware.TAxisToolCenter.T_CtrleSingle.xExecute) AND xMicroRodActive) OR NOT(xMicroRodActive)) ;
				xTmp:=	xTmp AND T_Station.THardware.TAxisToolRight.T_CtrleSingle.xDone
						AND T_Station.THardware.TAxisToolRight.T_CtrleSingle.xNotMoving
						AND NOT(T_Station.THardware.TAxisToolRight.T_CtrleSingle.xErr)
						AND NOT(T_Station.THardware.TAxisToolRight.T_CtrleSingle.xExecute);
				xTmp:=	xTmp AND T_Station.THardware.TAxisToolFeeder.T_CtrleSingle.xDone
						AND T_Station.THardware.TAxisToolFeeder.T_CtrleSingle.xNotMoving
						AND NOT(T_Station.THardware.TAxisToolFeeder.T_CtrleSingle.xErr)
						AND NOT(T_Station.THardware.TAxisToolFeeder.T_CtrleSingle.xExecute);
				xTmp:=	xTmp AND T_Station.THardware.TAxisGrindFeeder.T_CtrleSingle.xDone
						AND T_Station.THardware.TAxisGrindFeeder.T_CtrleSingle.xNotMoving
						AND NOT(T_Station.THardware.TAxisGrindFeeder.T_CtrleSingle.xErr)
						AND NOT(T_Station.THardware.TAxisGrindFeeder.T_CtrleSingle.xExecute);
				(* Start/Stop position or speed of teachin page has to be confirmed *)
				IF xTmp THEN
					iStepAction:=10;
				END_IF
			ELSE
				iStepAction:=95;
			END_IF;
		(* activ function axis *)
		10:	bStateMachine:=2;
			xSetStateMachine:=TRUE;
			xTmp:=	T_Station.THardware.TAxisToolLeft.T_CtrleSingle.xPower AND
					((T_Station.THardware.TAxisToolCenter.T_CtrleSingle.xPower AND xMicroRodActive) OR NOT(xMicroRodActive)) AND
					T_Station.THardware.TAxisToolRight.T_CtrleSingle.xPower AND
					T_Station.THardware.TAxisToolFeeder.T_CtrleSingle.xPower AND
					T_Station.THardware.TAxisGrindFeeder.T_CtrleSingle.xPower;
			IF xTmp THEN
				T_Station.THardware.TAxisToolLeft.T_CtrleSingle.iFunction:=4;
				IF xMicroRodActive THEN
					T_Station.THardware.TAxisToolCenter.T_CtrleSingle.iFunction:=4;
				END_IF;
				T_Station.THardware.TAxisToolRight.T_CtrleSingle.iFunction:=4;
				T_Station.THardware.TAxisToolFeeder.T_CtrleSingle.iFunction:=4;
				T_Station.THardware.TAxisGrindFeeder.T_CtrleSingle.iFunction:=4;
			ELSE
				IF NOT(T_Station.THardware.TAxisToolLeft.T_CtrleSingle.xPower) THEN
					T_Station.THardware.TAxisToolLeft.T_CtrleSingle.iFunction:=3;
				END_IF;
				IF xMicroRodActive THEN
					IF NOT(T_Station.THardware.TAxisToolCenter.T_CtrleSingle.xPower) THEN
						T_Station.THardware.TAxisToolCenter.T_CtrleSingle.iFunction:=3;
					END_IF;
				END_IF;
				IF NOT(T_Station.THardware.TAxisToolRight.T_CtrleSingle.xPower) THEN
					T_Station.THardware.TAxisToolRight.T_CtrleSingle.iFunction:=3;
				END_IF;
				IF NOT(T_Station.THardware.TAxisToolFeeder.T_CtrleSingle.xPower) THEN
					T_Station.THardware.TAxisToolFeeder.T_CtrleSingle.iFunction:=3;
				END_IF;
				IF NOT(T_Station.THardware.TAxisGrindFeeder.T_CtrleSingle.xPower) THEN
					T_Station.THardware.TAxisGrindFeeder.T_CtrleSingle.iFunction:=3;
				END_IF;
			END_IF;
			T_Station.THardware.TAxisToolLeft.T_CtrleSingle.xExecute:=TRUE;
			T_Station.THardware.TAxisToolCenter.T_CtrleSingle.xExecute:=xMicroRodActive;
			T_Station.THardware.TAxisToolRight.T_CtrleSingle.xExecute:=TRUE;
			T_Station.THardware.TAxisToolFeeder.T_CtrleSingle.xExecute:=TRUE;
			T_Station.THardware.TAxisGrindFeeder.T_CtrleSingle.xExecute:=TRUE;
			(* next step *)
			iStepAction:=20;
			xStepActionDone:=FALSE;
		(* confirm execution *)
		20:	IF NOT(xStepActionDone) THEN
			(* confirm execution *)
				T_Station.THardware.TAxisToolLeft.T_CtrleSingle.xExecute:=FALSE;
				T_Station.THardware.TAxisToolCenter.T_CtrleSingle.xExecute:=FALSE;
				T_Station.THardware.TAxisToolRight.T_CtrleSingle.xExecute:=FALSE;
				T_Station.THardware.TAxisToolFeeder.T_CtrleSingle.xExecute:=FALSE;
				T_Station.THardware.TAxisGrindFeeder.T_CtrleSingle.xExecute:=FALSE;
				xStepActionDone:=TRUE;
			ELSE
				xTmp:=	T_Station.THardware.TAxisToolLeft.T_CtrleSingle.xDone AND
						((T_Station.THardware.TAxisToolCenter.T_CtrleSingle.xDone AND xMicroRodActive) OR NOT(xMicroRodActive)) AND
						T_Station.THardware.TAxisToolRight.T_CtrleSingle.xDone AND
						T_Station.THardware.TAxisToolFeeder.T_CtrleSingle.xDone AND
						T_Station.THardware.TAxisGrindFeeder.T_CtrleSingle.xDone;
				IF xTmp THEN
				(* confirm action next step *)
					bStateMachine:=1;
					xSetStateMachine:=TRUE;
					iStepAction:=90;
					xStepActionDone:=FALSE;
				ELSE
					xTmp:=	T_Station.THardware.TAxisToolLeft.T_CtrleSingle.xErr OR
							(T_Station.THardware.TAxisToolCenter.T_CtrleSingle.xErr AND xMicroRodActive) OR
							T_Station.THardware.TAxisToolRight.T_CtrleSingle.xErr OR
							T_Station.THardware.TAxisToolFeeder.T_CtrleSingle.xErr OR
							T_Station.THardware.TAxisGrindFeeder.T_CtrleSingle.xErr;
					IF xTmp THEN
					(* activ action not ready or error *)
						iStepAction:=99;
						xStepActionDone:=FALSE;
					END_IF
				END_IF
			END_IF
		(* action done *)
		90:	T_Visu.ptrT_ExchgParam^.T_StationCommon.wState:=T_Visu.ptrT_ExchgParam^.T_StationCommon.wState AND 16#BF;
			T_Visu.T_CtrleAction.xDone:=TRUE;
			T_Visu.T_CtrleAction.xNotReady:=FALSE;
			T_Visu.T_CtrleAction.xErr:=FALSE;
			T_Visu.T_CtrleAction.udiErrorID:=0;
			xToggleAllAxisPower:=FALSE;
		(* axis not ready *)
		95:	T_Visu.ptrT_ExchgParam^.T_StationCommon.wState:=T_Visu.ptrT_ExchgParam^.T_StationCommon.wState AND 16#BF;
			TimerNotReady(IN:=TRUE);
			xToggleAllAxisPower:=FALSE;
		(* error *)
		99:	T_Visu.ptrT_ExchgParam^.T_StationCommon.wState:=T_Visu.ptrT_ExchgParam^.T_StationCommon.wState AND 16#BF;
			T_Visu.T_CtrleAction.xDone:=TRUE;
			T_Visu.T_CtrleAction.xNotReady:=FALSE;
			diErrorNr:=0;
			IF T_Station.THardware.TAxisToolLeft.T_CtrleSingle.xErr THEN
				diErrorNr:=1000000 + T_Station.THardware.TAxisToolLeft.T_CtrleSingle.udiErrorID;
			END_IF;
			IF xMicroRodActive THEN
				IF T_Station.THardware.TAxisToolCenter.T_CtrleSingle.xErr THEN
					diErrorNr:=2000000 + T_Station.THardware.TAxisToolCenter.T_CtrleSingle.udiErrorID;
				END_IF;
			END_IF;
			IF T_Station.THardware.TAxisToolRight.T_CtrleSingle.xErr THEN
				diErrorNr:=3000000 + T_Station.THardware.TAxisToolRight.T_CtrleSingle.udiErrorID;
			END_IF;
			IF T_Station.THardware.TAxisToolFeeder.T_CtrleSingle.xErr THEN
				diErrorNr:=4000000 + T_Station.THardware.TAxisToolFeeder.T_CtrleSingle.udiErrorID;
			END_IF;
			IF T_Station.THardware.TAxisGrindFeeder.T_CtrleSingle.xErr THEN
				diErrorNr:=5000000 + T_Station.THardware.TAxisGrindFeeder.T_CtrleSingle.udiErrorID;
			END_IF;
			FBErrorMessage(	diErrorNr:=diErrorNr,
							T_ErrorList:=T_ErrorList);
			T_Visu.ptrT_ExchgParam^.T_Visu.T_Message.sDynamicTextEnglish:=FBErrorMessage.sErrorTextEnglish;
			T_Visu.ptrT_ExchgParam^.T_Visu.T_Message.sDynamicTextDeutsch:=FBErrorMessage.sErrorTextDeutsch;
			T_Visu.ptrT_ExchgParam^.T_Visu.T_Message.sDynamicTextFrancais:=FBErrorMessage.sErrorTextFrancais;
			T_Visu.ptrT_ExchgParam^.T_SafetyCtrl.xSetForceError:=TRUE;
			T_Visu.ptrT_ExchgParam^.T_SafetyCtrl.diSetForceErrorNr:=diErrorNr;
			T_Visu.T_CtrleAction.xErr:=FALSE;
			T_Visu.T_CtrleAction.udiErrorID:=0;
			T_Station.THardware.TAxisToolLeft.T_CtrleSingle.iFunction:=1;
			T_Station.THardware.TAxisToolLeft.T_CtrleSingle.xExecute:=T_Station.THardware.TAxisToolLeft.T_CtrleSingle.xErr;
			IF xMicroRodActive THEN
				T_Station.THardware.TAxisToolCenter.T_CtrleSingle.iFunction:=1;
				T_Station.THardware.TAxisToolCenter.T_CtrleSingle.xExecute:=T_Station.THardware.TAxisToolCenter.T_CtrleSingle.xErr;
			END_IF;
			T_Station.THardware.TAxisToolRight.T_CtrleSingle.iFunction:=1;
			T_Station.THardware.TAxisToolRight.T_CtrleSingle.xExecute:=T_Station.THardware.TAxisToolRight.T_CtrleSingle.xErr;
			T_Station.THardware.TAxisToolFeeder.T_CtrleSingle.iFunction:=1;
			T_Station.THardware.TAxisToolFeeder.T_CtrleSingle.xExecute:=T_Station.THardware.TAxisToolFeeder.T_CtrleSingle.xErr;
			T_Station.THardware.TAxisGrindFeeder.T_CtrleSingle.iFunction:=1;
			T_Station.THardware.TAxisGrindFeeder.T_CtrleSingle.xExecute:=T_Station.THardware.TAxisGrindFeeder.T_CtrleSingle.xErr;
			xToggleAllAxisPower:=FALSE;
		END_CASE
	END_IF

(* Correction Tool Diameter +,++,-,-- *)
	IF xCorrectionToolDiameterAdd OR xCorrectionToolDiameterAddMore OR 	xCorrectionToolDiameterSub OR xCorrectionToolDiameterSubMore OR xResetToolDiameterCorrection OR xKeyPadActivation THEN
		CASE iStepAction OF
		(* check visu *)
		1:	xTmp:=	TRUE;
			IF xTmp THEN
				(* next Step *)
				iStepAction :=10;
				IF xResetToolDiameterCorrection THEN
					(* next Step *)
					iStepAction :=20;
				END_IF;
				IF xKeyPadActivation THEN
					IF (T_Visu.T_PlcParam.dwActualPage = 420) OR (T_Visu.T_PlcParam.dwActualPage = 11) OR (T_Visu.T_PlcParam.dwActualPage = 21) THEN
						(* next Step *)
						iStepAction :=30;
					END_IF;
					IF (T_Visu.T_PlcParam.dwActualPage = 430) THEN
						(* next Step *)
						iStepAction :=40;
					END_IF;
				END_IF;
			(* activ error *)
			ELSE iStepAction:=95; END_IF
		10:	IF xCorrectionToolDiameterAdd THEN
				rCorrectionValue:=0.1;
			END_IF;
			IF xCorrectionToolDiameterAddMore THEN
				rCorrectionValue:=1.0;
			END_IF;
			IF xCorrectionToolDiameterSub THEN
				rCorrectionValue:=-0.1;
			END_IF;
			IF xCorrectionToolDiameterSubMore THEN
				rCorrectionValue:=-1.0;
			END_IF;
			T_Visu.ptrT_ExchgParam^.T_InfoValueCommon.rCorrectionToolDiameter:=T_Visu.ptrT_ExchgParam^.T_InfoValueCommon.rCorrectionToolDiameter + rCorrectionValue;
			IF (T_Visu.ptrT_ExchgParam^.T_InfoValueCommon.rCorrectionToolDiameter < 0.1) AND
			    (T_Visu.ptrT_ExchgParam^.T_InfoValueCommon.rCorrectionToolDiameter > -0.1) THEN
				T_Visu.ptrT_ExchgParam^.T_InfoValueCommon.rCorrectionToolDiameter:=0.0;
			END_IF;
			(* next Step *)
			iStepAction :=90;
		20:	T_Visu.ptrT_ExchgParam^.T_InfoValueCommon.rCorrectionToolDiameter:=0.0;
			(* next Step *)
			iStepAction :=90;
		30:	T_Visu.ptrT_ExchgParam^.T_InfoValueCommon.xKeyPadActivation:=NOT(T_Visu.ptrT_ExchgParam^.T_InfoValueCommon.xKeyPadActivation);
			(* next Step *)
			iStepAction :=90;
		40:	(* 0= 3 value prisma, 1 = 3 value prisma input para, 2 = 2 value prisma, 3 = 2 value prisma input para *)
			IF (T_Visu.ptrT_ExchgParam^.T_StationCommon.T_PrismPara.bStateInputPrisma = 0) THEN
				T_Visu.ptrT_ExchgParam^.T_StationCommon.T_PrismPara.bStateInputPrisma:=1;
			ELSIF (T_Visu.ptrT_ExchgParam^.T_StationCommon.T_PrismPara.bStateInputPrisma = 1) THEN
				T_Visu.ptrT_ExchgParam^.T_StationCommon.T_PrismPara.bStateInputPrisma:=0;
			ELSIF (T_Visu.ptrT_ExchgParam^.T_StationCommon.T_PrismPara.bStateInputPrisma = 2) THEN
				T_Visu.ptrT_ExchgParam^.T_StationCommon.T_PrismPara.bStateInputPrisma:=3;
			ELSIF (T_Visu.ptrT_ExchgParam^.T_StationCommon.T_PrismPara.bStateInputPrisma = 3) THEN
				T_Visu.ptrT_ExchgParam^.T_StationCommon.T_PrismPara.bStateInputPrisma:=2;
			END_IF;
			(* next Step *)
			iStepAction:=90;
		(* change page done *)
		90:	T_Visu.T_CtrleAction.xDone:=TRUE;
			T_Visu.T_CtrleAction.xNotReady:=FALSE;
			T_Visu.T_CtrleAction.xErr:=FALSE;
			T_Visu.T_CtrleAction.udiErrorID:=0;
			xCorrectionToolDiameterAdd:=xCorrectionToolDiameterAddMore:=xCorrectionToolDiameterSub:=xCorrectionToolDiameterSubMore:=xResetToolDiameterCorrection:=xKeyPadActivation:=FALSE;
		(* not ready *)
		95:	T_Visu.T_CtrleAction.xDone:=TRUE;
			T_Visu.T_CtrleAction.xNotReady:=FALSE;
			T_Visu.T_CtrleAction.xErr:=FALSE;
			T_Visu.T_CtrleAction.udiErrorID:=0;
			xCorrectionToolDiameterAdd:=xCorrectionToolDiameterAddMore:=xCorrectionToolDiameterSub:=xCorrectionToolDiameterSubMore:=xResetToolDiameterCorrection:=xKeyPadActivation:=FALSE;
		END_CASE
	END_IF;

(* Function Correction Tool Diameter *)
	IF xFctCorrectionToolDiameter THEN
		CASE iStepAction OF
		(* check axis *)
		1:	IF NOT T_Station.TControl.xHardwareConfigError THEN
				xStepActionDone:=FALSE;
				iStepAction:=95;
				xTmp:=	T_Station.THardware.TAxisGrindFeeder.T_CtrleSingle.xDone
						AND T_Station.THardware.TAxisGrindFeeder.T_CtrleSingle.xReady
						AND T_Station.THardware.TAxisGrindFeeder.T_CtrleSingle.xNotMoving
						AND NOT(T_Station.THardware.TAxisGrindFeeder.T_CtrleSingle.xErr)
						AND NOT(T_Station.THardware.TAxisGrindFeeder.T_CtrleSingle.xExecute);
				(* Start/Stop position or speed of teachin page has to be confirmed *)
				IF xTmp THEN
					iStepAction:=10;
				END_IF
			ELSE
				iStepAction:=95;
			END_IF;
		(* Display message to ask for confirmation *)
		10:	T_Visu.ptrT_ExchgParam^.T_Visu.T_Message.iState:=108;
			iStepAction:=20;
		(* waiting for key <Enter> or <Esc> *)
		20:	IF RisingEdgeKeyPanel_Enter.Q THEN iStepAction:=30;
			ELSE IF RisingEdgeKeyPanel_Esc.Q THEN iStepAction:=90; END_IF END_IF
			(* An other message has been displayed, stop teach action *)
			IF T_Visu.ptrT_ExchgParam^.T_Visu.T_Message.iState<>108 THEN iStepAction:=90; END_IF
		(* activ function axis *)
		30:	(*T_Visu.ptrT_ExchgParam^.T_InfoValueCommon.rActualGrindAxisPosition:=T_Visu.ptrT_ExchgParam^.T_InfoValueCommon.rActualGrindAxisPosition - T_Visu.ptrT_ExchgParam^.T_InfoValueCommon.rCorrectionToolDiameter;*)
			T_Station.THardware.TAxisGrindFeeder.T_CtrleSingle.rSetPosition:=T_Station.THardware.TAxisGrindFeeder.T_LiveValue.lrActualPosition - T_Visu.ptrT_ExchgParam^.T_InfoValueCommon.rCorrectionToolDiameter;
			T_Visu.ptrT_ExchgParam^.T_InfoValueCommon.rCorrectionToolDiameter:=0.0;
			T_Station.THardware.TAxisGrindFeeder.T_CtrleSingle.iFunction:=11;
			T_Station.THardware.TAxisGrindFeeder.T_CtrleSingle.xExecute:=TRUE;
			(* next step *)
			iStepAction:=50;
			xStepActionDone:=FALSE;
		(* confirm execution *)
		50:	IF NOT(xStepActionDone) THEN
			(* confirm execution *)
				T_Station.THardware.TAxisGrindFeeder.T_CtrleSingle.xExecute:=FALSE;
				xStepActionDone:=TRUE;
			ELSE
				IF T_Station.THardware.TAxisGrindFeeder.T_CtrleSingle.xDone THEN
				(* confirm action next step *)
					iStepAction:=90;
					xStepActionDone:=FALSE;
				ELSE
					IF T_Station.THardware.TAxisGrindFeeder.T_CtrleSingle.xErr THEN
					(* activ action not ready or error *)
						iStepAction:=99;
						xStepActionDone:=FALSE;
					END_IF
				END_IF
			END_IF
		(* action done *)
		90:	T_Visu.ptrT_ExchgParam^.T_StationCommon.wState:=T_Visu.ptrT_ExchgParam^.T_StationCommon.wState AND 16#BF;
			T_Visu.T_CtrleAction.xDone:=TRUE;
			T_Visu.T_CtrleAction.xNotReady:=FALSE;
			T_Visu.T_CtrleAction.xErr:=FALSE;
			T_Visu.T_CtrleAction.udiErrorID:=0;
			xFctCorrectionToolDiameter:=FALSE;
		(* axis not ready *)
		95:	T_Visu.ptrT_ExchgParam^.T_StationCommon.wState:=T_Visu.ptrT_ExchgParam^.T_StationCommon.wState AND 16#BF;
			TimerNotReady(IN:=TRUE);
			xFctCorrectionToolDiameter:=FALSE;
		(* error *)
		99:	T_Visu.ptrT_ExchgParam^.T_StationCommon.wState:=T_Visu.ptrT_ExchgParam^.T_StationCommon.wState AND 16#BF;
			T_Visu.T_CtrleAction.xDone:=TRUE;
			T_Visu.T_CtrleAction.xNotReady:=FALSE;
			IF (T_Station.THardware.TAxisGrindFeeder.T_Config_Gen.iTyp <> 0) THEN
				diErrorNr:=(T_Station.THardware.TAxisGrindFeeder.T_Config_Gen.iTyp * 1000000) + T_Station.THardware.TAxisGrindFeeder.T_CtrleSingle.udiErrorID;
			ELSE
				diErrorNr:=0;
			END_IF;
			FBErrorMessage(	diErrorNr:=diErrorNr,
							T_ErrorList:=T_ErrorList);
			T_Visu.ptrT_ExchgParam^.T_Visu.T_Message.sDynamicTextEnglish:=FBErrorMessage.sErrorTextEnglish;
			T_Visu.ptrT_ExchgParam^.T_Visu.T_Message.sDynamicTextDeutsch:=FBErrorMessage.sErrorTextDeutsch;
			T_Visu.ptrT_ExchgParam^.T_Visu.T_Message.sDynamicTextFrancais:=FBErrorMessage.sErrorTextFrancais;
			T_Visu.ptrT_ExchgParam^.T_SafetyCtrl.xSetForceError:=TRUE;
			T_Visu.ptrT_ExchgParam^.T_SafetyCtrl.diSetForceErrorNr:=diErrorNr;
			T_Visu.T_CtrleAction.xErr:=FALSE;
			T_Visu.T_CtrleAction.udiErrorID:=0;
			T_Station.THardware.TAxisGrindFeeder.T_CtrleSingle.iFunction:=1;
			T_Station.THardware.TAxisGrindFeeder.T_CtrleSingle.xExecute:=TRUE;
			xFctCorrectionToolDiameter:=FALSE;
		END_CASE
	END_IF;

(* Select Prisma 1 or 2 Input *)
	IF xSelectPrisma THEN
		CASE iStepAction OF
		(* check visu *)
		1:	xTmp:=	TRUE;
			IF xTmp THEN
				(* next Step *)
				iStepAction :=10;
			(* activ error *)
			ELSE iStepAction:=95; END_IF
		10:	(* 0= 3 value prisma, 1 = 3 value prisma input para, 2 = 2 value prisma, 3 = 2 value prisma input para *)
			IF (T_Visu.ptrT_ExchgParam^.T_StationCommon.T_PrismPara.bStateInputPrisma = 0) OR (T_Visu.ptrT_ExchgParam^.T_StationCommon.T_PrismPara.bStateInputPrisma = 1) THEN
				T_Visu.ptrT_ExchgParam^.T_StationCommon.T_PrismPara.bStateInputPrisma:=2;
			ELSIF (T_Visu.ptrT_ExchgParam^.T_StationCommon.T_PrismPara.bStateInputPrisma = 2) OR (T_Visu.ptrT_ExchgParam^.T_StationCommon.T_PrismPara.bStateInputPrisma = 3) THEN
				T_Visu.ptrT_ExchgParam^.T_StationCommon.T_PrismPara.bStateInputPrisma:=0;
			END_IF;
			(* next Step *)
			iStepAction:=90;
		(* change page done *)
		90:	T_Visu.T_CtrleAction.xDone:=TRUE;
			T_Visu.T_CtrleAction.xNotReady:=FALSE;
			T_Visu.T_CtrleAction.xErr:=FALSE;
			T_Visu.T_CtrleAction.udiErrorID:=0;
			xSelectPrisma:=FALSE;
		(* not ready *)
		95:	T_Visu.T_CtrleAction.xDone:=TRUE;
			T_Visu.T_CtrleAction.xNotReady:=FALSE;
			T_Visu.T_CtrleAction.xErr:=FALSE;
			T_Visu.T_CtrleAction.udiErrorID:=0;
			xSelectPrisma:=FALSE;
		END_CASE
	END_IF;

(* Set calculated ToolRotation Torque *)
	IF xSetCalculToolRotTorque THEN
		CASE iStepAction OF
		(* check visu *)
		1:	xTmp:=	TRUE;
			IF xTmp THEN
				(* next Step *)
				iStepAction :=10;
			(* activ error *)
			ELSE iStepAction:=95; END_IF
		10:	uiToolLeftZeroTorque:=T_Station.THardware.TAxisToolLeft.T_LiveValue.uiActualTorque;
			FBCalcTorqueToolLeft(	xStart:=TRUE,
									uiActualTorque:= T_Station.THardware.TAxisToolLeft.T_LiveValue.uiActualTorque,
									uiZeroTorque:=uiToolLeftZeroTorque,
									iStepCalc:= 100);
			uiToolCenterZeroTorque:=T_Station.THardware.TAxisToolCenter.T_LiveValue.uiActualTorque;
			FBCalcTorqueToolCenter(	xStart:=TRUE,
									uiActualTorque:= T_Station.THardware.TAxisToolCenter.T_LiveValue.uiActualTorque,
									uiZeroTorque:=uiToolCenterZeroTorque,
									iStepCalc:= 100);
			uiToolRightZeroTorque:=T_Station.THardware.TAxisToolRight.T_LiveValue.uiActualTorque;
			FBCalcTorqueToolRight(	xStart:=TRUE,
									uiActualTorque:= T_Station.THardware.TAxisToolRight.T_LiveValue.uiActualTorque,
									uiZeroTorque:=uiToolRightZeroTorque,
									iStepCalc:= 100);
			(* next Step *)
			iStepAction:=90;
		(* change page done *)
		90:	T_Visu.T_CtrleAction.xDone:=TRUE;
			T_Visu.T_CtrleAction.xNotReady:=FALSE;
			T_Visu.T_CtrleAction.xErr:=FALSE;
			T_Visu.T_CtrleAction.udiErrorID:=0;
			xSetCalculToolRotTorque:=FALSE;
		(* not ready *)
		95:	T_Visu.T_CtrleAction.xDone:=TRUE;
			T_Visu.T_CtrleAction.xNotReady:=FALSE;
			T_Visu.T_CtrleAction.xErr:=FALSE;
			T_Visu.T_CtrleAction.udiErrorID:=0;
			xSetCalculToolRotTorque:=FALSE;
		END_CASE
	END_IF;

(* Reset calculated ToolRotation Torque *)
	IF xResetCalculToolRotTorque THEN
		CASE iStepAction OF
		(* check visu *)
		1:	xTmp:=	TRUE;
			IF xTmp THEN
				(* next Step *)
				iStepAction :=10;
			(* activ error *)
			ELSE iStepAction:=95; END_IF
		10:	uiToolLeftZeroTorque:=0;
			FBCalcTorqueToolLeft(	xStart:=TRUE,
									uiActualTorque:= T_Station.THardware.TAxisToolLeft.T_LiveValue.uiActualTorque,
									uiZeroTorque:=uiToolLeftZeroTorque,
									iStepCalc:= 100);
			uiToolCenterZeroTorque:=0;
			FBCalcTorqueToolCenter(	xStart:=TRUE,
									uiActualTorque:= T_Station.THardware.TAxisToolCenter.T_LiveValue.uiActualTorque,
									uiZeroTorque:=uiToolCenterZeroTorque,
									iStepCalc:= 100);
			uiToolRightZeroTorque:=0;
			FBCalcTorqueToolRight(	xStart:=TRUE,
									uiActualTorque:= T_Station.THardware.TAxisToolRight.T_LiveValue.uiActualTorque,
									uiZeroTorque:=uiToolRightZeroTorque,
									iStepCalc:= 100);
			(* next Step *)
			iStepAction:=90;
		(* change page done *)
		90:	T_Visu.T_CtrleAction.xDone:=TRUE;
			T_Visu.T_CtrleAction.xNotReady:=FALSE;
			T_Visu.T_CtrleAction.xErr:=FALSE;
			T_Visu.T_CtrleAction.udiErrorID:=0;
			xResetCalculToolRotTorque:=FALSE;
		(* not ready *)
		95:	T_Visu.T_CtrleAction.xDone:=TRUE;
			T_Visu.T_CtrleAction.xNotReady:=FALSE;
			T_Visu.T_CtrleAction.xErr:=FALSE;
			T_Visu.T_CtrleAction.udiErrorID:=0;
			xResetCalculToolRotTorque:=FALSE;
		END_CASE
	END_IF;

(* Switch WireFeed Jog Speed Slow/Fast *)
	IF xSlowFastJogToolRotation OR xSlowFastJogToolFeeder OR xSlowFastJogGrindFeeder THEN
		CASE iStepAction OF
		(* check visu *)
		1:	xTmp:=	TRUE;
			IF xTmp THEN
				(* next Step *)
				iStepAction :=10;
			(* activ error *)
			ELSE iStepAction:=95; END_IF
		10:	IF xSlowFastJogToolRotation THEN
				T_Visu.ptrT_ExchgParam^.T_TeachIn.xSlowFastToolRotation:=NOT(T_Visu.ptrT_ExchgParam^.T_TeachIn.xSlowFastToolRotation);
			END_IF;
			IF xSlowFastJogToolFeeder THEN
				T_Visu.ptrT_ExchgParam^.T_TeachIn.xSlowFastToolFeed:=NOT(T_Visu.ptrT_ExchgParam^.T_TeachIn.xSlowFastToolFeed);
			END_IF;
			IF xSlowFastJogGrindFeeder THEN
				T_Visu.ptrT_ExchgParam^.T_TeachIn.xSlowFastGrindFeeder:=NOT(T_Visu.ptrT_ExchgParam^.T_TeachIn.xSlowFastGrindFeeder);
			END_IF;
			(* next Step *)
			iStepAction:=90;
		(* change page done *)
		90:	T_Visu.T_CtrleAction.xDone:=TRUE;
			T_Visu.T_CtrleAction.xNotReady:=FALSE;
			T_Visu.T_CtrleAction.xErr:=FALSE;
			T_Visu.T_CtrleAction.udiErrorID:=0;
			xSlowFastJogToolRotation:=xSlowFastJogToolFeeder:=xSlowFastJogGrindFeeder:=FALSE;
		(* not ready *)
		95:	T_Visu.T_CtrleAction.xDone:=TRUE;
			T_Visu.T_CtrleAction.xNotReady:=FALSE;
			T_Visu.T_CtrleAction.xErr:=FALSE;
			T_Visu.T_CtrleAction.udiErrorID:=0;
			xSlowFastJogToolRotation:=xSlowFastJogToolFeeder:=xSlowFastJogGrindFeeder:=FALSE;
		END_CASE
	END_IF;



VisuFunction_Axis;
VisuFunction_AxisTeach;
VisuFunction_Cylinder;
VisuFunction_StationFunction;
VisuFunction_SetupSection;
VisuFunction_ProfileManagement;
VisuFunction_NovRAM;
VisuFunction_ProcessFunction;
CtrlProcessFunction;
VisuFunction_ProcessStop;
VisuFunction_SetupWarmup;
VisuFunction_SpecialFunction;



(************************************************************************************************************************************************************************)
(***************                                                 management for the changement of a page on the visualisation                                                 ********************)
(************************************************************************************************************************************************************************)
(* waiting for changing page *)
	RisingEdgeExecute(CLK:=T_Visu.T_CtrleVisu.xExecute);
	IF RisingEdgeExecute.Q THEN
		CASE T_Visu.T_CtrleVisu.iFunction OF
		(* change page *)
		1:	xChangePage:=TRUE;
			dwInCount_QVisCmd:=T_CtrleQVis.dwInCount;
		ELSE
		(* function not implemented *)
			T_Visu.T_CtrleVisu.xDone:=FALSE;
			T_Visu.T_CtrleVisu.xErr:=TRUE;
			T_Visu.T_CtrleVisu.udiErrorID:=16#F000;
		END_CASE
		(* Init. variable *)
		T_Visu.T_CtrleVisu.xDone:=FALSE;
		T_Visu.T_CtrleVisu.xErr:=FALSE;
		T_Visu.T_CtrleVisu.udiErrorID:=0;
		(* exit FB *)
		RETURN;
	END_IF

(* waiting for changing page from the PLC *)
	IF xChangePage THEN
		IF dwInCount_QVisCmd = T_CtrleQVis.dwInCount THEN
			(* Init. command *)
			T_CtrleQVis.dwInCommand:=1;
			T_CtrleQVis.dwInQVisCtrlAddress:=ADR(T_CtrleQVis);
			T_CtrleQVis.dwInParameterAddress:=ADR(T_Visu.T_PlcParam.dwSetNewPage);
			(* start command *)
			T_CtrleQVis.dwInCount:=T_CtrleQVis.dwInCount+1;
		ELSE
			IF T_CtrleQVis.dwInCount = T_CtrleQVis.dwOutCount THEN
			(* command done *)
				T_Visu.T_CtrleVisu.xExecute:=FALSE;
				IF T_CtrleQVis.diOutStatus = 0 THEN
				(* command done without error *)
					T_Visu.T_CtrleVisu.xDone:=TRUE;
					T_Visu.T_CtrleVisu.xErr:=FALSE;
					T_Visu.T_CtrleVisu.udiErrorID:=0;
					(* update value *)
					T_Visu.T_PlcParam.dwPreviousPage:=T_Visu.T_PlcParam.dwActualPage;
					T_Visu.T_PlcParam.dwActualPage:=T_Visu.T_PlcParam.dwSetNewPage;
					IF (T_Visu.T_PlcParam.dwActualPage = 10) THEN
						wNormalLayerActivTask:=1;
						wNormalLayerActivPage:=10;
					END_IF;
				ELSE
				(* command done with error *)
					T_Visu.T_CtrleVisu.xDone:=FALSE;
					T_Visu.T_CtrleVisu.xErr:=TRUE;
					T_Visu.T_CtrleVisu.udiErrorID:=16#F400 + DINT_TO_UDINT(T_CtrleQVis.diOutStatus);
				END_IF
				(* reset variable 'xChangePage' *)
				xChangePage:=FALSE;
			END_IF
		END_IF
	END_IF
END_FUNCTION_BLOCK
ACTION CtrlFunctionButton:
(* Managment Bt Function panel *)
	IF (T_Visu.T_PlcParam.dwActualPage = 10) OR (T_Visu.T_PlcParam.dwActualPage = 110) THEN
		IF NOT(xMicroRodActive) THEN
		(* For MicroWire no Function for move the ToolFeeder to the StartPos-->Cancel Function F5 *)
			wMaskFunctionPanel:=wMaskFunctionPanel AND 16#FFEF;
			T_Visu.ptrT_ExchgParam^.T_BtFunctionPanel.wNotMasktext:=T_Visu.ptrT_ExchgParam^.T_BtFunctionPanel.wNotMasktext OR 16#10;
		END_IF;
	END_IF;
	IF (T_Visu.T_PlcParam.dwActualPage = 20) THEN
		IF NOT(xMicroRodActive) THEN
		(* For MicroWire no Function for move the ToolFeeder to the StartPos-->Cancel Function F5 *)
			wMaskFunctionPanel:=wMaskFunctionPanel AND 16#FFEF;
			T_Visu.ptrT_ExchgParam^.T_BtFunctionPanel.wNotMasktext:=T_Visu.ptrT_ExchgParam^.T_BtFunctionPanel.wNotMasktext OR 16#10;
		END_IF;
	END_IF;
	IF (T_Visu.T_PlcParam.dwActualPage = 310) THEN
		IF NOT(xMicroRodActive) THEN
		(* For MicroWire no Function for no Position to save for ToolFeeder-->Cancel Function F3 and F6 *)
			wMaskFunctionPanel:=wMaskFunctionPanel AND 16#FFDB;
			T_Visu.ptrT_ExchgParam^.T_BtFunctionPanel.wNotMasktext:=T_Visu.ptrT_ExchgParam^.T_BtFunctionPanel.wNotMasktext OR 16#24;
		END_IF;
	END_IF;
	IF (T_Visu.T_PlcParam.dwActualPage = 320) THEN
		IF NOT(xMicroRodActive) THEN
		(* For MicroWire no Function for ToolFeeder-->Cancel Function F1, F2, F3 and F4 *)
			wMaskFunctionPanel:=wMaskFunctionPanel AND 16#0;
			T_Visu.ptrT_ExchgParam^.T_BtFunctionPanel.wNotMasktext:=T_Visu.ptrT_ExchgParam^.T_BtFunctionPanel.wNotMasktext OR 16#FFFF;
		END_IF;
	END_IF;



	IF (wForceMaskFunctionPanel <> 0) THEN	(* IGS *)
		(* Wurde von einer Funktion überschrieben *)
		T_ConfigPage.wMaskFunctionPanel:=wForceMaskFunctionPanel;
		wMaskFunctionPanel:=wForceMaskFunctionPanel;
		wForceMaskFunctionPanel:=0;
	END_IF;
	FOR ii:=1 TO 12 DO
		IF (aiForceRTrigActionFunctionPanel[ii] <> 0) THEN
			(* Wurde von einer Funktion überschrieben *)
			T_ConfigPage.aiRTrigActionFunctionPanel:=aiForceRTrigActionFunctionPanel;
			EXIT;
		END_IF;
	END_FOR;
	aiForceRTrigActionFunctionPanel:=aiDelectRTrigActionFunctionPanel;



	RisingEdgeBtFunctionPanel(CLK:=(T_Visu.ptrT_ExchgParam^.T_BtFunctionPanel.wActivBt AND wMaskFunctionPanel) <> 16#0);
	FallingEdgeBtFunctionPanel(CLK:=(T_Visu.ptrT_ExchgParam^.T_BtFunctionPanel.wActivBt AND wMaskFunctionPanel) <> 16#0);
	xTmp:=	NOT(xChangePage)
			AND T_Visu.T_CtrleAction.xDone
			AND NOT(T_Visu.T_CtrleAction.xExecute)
			AND NOT(T_StartUp.T_State.xBlockChangeMovementVisu);
	IF xTmp THEN
		(* Rising edge action *)
		IF RisingEdgeBtFunctionPanel.Q THEN
		(* Init. variable *)
			ii:=1;
			wTmp:=T_Visu.ptrT_ExchgParam^.T_BtFunctionPanel.wActivBt;
			WHILE wTmp <> 16#0 DO
				IF (wTmp AND 16#1) = 16#1 THEN EXIT; END_IF
				wTmp:=ROR(wTmp,1);
				ii:=ii+1;
			END_WHILE
			(* set the new action if present *)
			IF  T_ConfigPage.aiRTrigActionFunctionPanel[ii] <> 0 THEN
				T_Visu.T_CtrleAction.iFunction:= T_ConfigPage.aiRTrigActionFunctionPanel[ii];
				T_Visu.T_CtrleAction.xExecute:=TRUE;
			END_IF
		END_IF
	END_IF
END_ACTION
ACTION CtrlPanelLeftButton:
(*Management Bt Panel left *)
	IF T_Visu.ptrT_ExchgParam^.T_Config.xNoTouchScreenBtPanel THEN
		wActivBtLeft:=wSPSSpecialButton;
	ELSE
		wActivBtLeft:=INT_TO_WORD(T_Visu.ptrT_ExchgParam^.T_TouchScreenBtPanel.iActivBtLeft);
	END_IF;
	RisingEdgeSpecialLayer(CLK:=xSecurityKey);
	FallingEdgeSpecialLayer(CLK:=xSecurityKey);
	RisingEdgeBtPanelLeft(CLK:=((wActivBtLeft AND wMaskBtPanelLeft) <> 16#0) AND T_Visu.ptrT_ExchgParam^.T_Visu.bActivSpecialLayer <> 0);
	FallingEdgeBtPanelLeft(CLK:=((wActivBtLeft AND wMaskBtPanelLeft) <> 16#0) AND T_Visu.ptrT_ExchgParam^.T_Visu.bActivSpecialLayer <> 0);
	xTmp:=	NOT(xChangePage)
			AND (T_Visu.T_CtrleAction.xDone OR ((xOverlayMeasureToolDia OR xOverlayGrindFeedSetPlung OR T_Visu.ptrT_ExchgParam^.T_FunctionCommon.xOpenOverlayMessageBox) AND FallingEdgeSpecialLayer.Q))
			AND NOT(T_Visu.T_CtrleAction.xExecute)
			AND NOT(T_StartUp.T_State.xBlockChangeMovementVisu)
			AND NOT(T_StartUp.T_State.xBlockVisuNavigation)
			AND T_StartUp.T_State.xCompleted;
	IF xTmp THEN
		IF RisingEdgeSpecialLayer.Q THEN
			CASE bOldActivSpecialLayer OF
				1:	T_Visu.ptrT_ExchgParam^.T_Visu.bActivSpecialLayer:=1;
					T_Visu.ptrT_ExchgParam^.T_TouchScreenBtPanel.iStateBtLeft:=1;
					T_Visu.ptrT_ExchgParam^.T_TouchScreenNavPanel.wState:=wSpecialLayerGeneralActivTask;
					ii:=1;
					wTmp:=wSpecialLayerGeneralActivTask;
					WHILE wTmp <> 16#0 DO
						IF (wTmp AND 16#1) = 16#1 THEN EXIT; END_IF
						wTmp:=ROR(wTmp,1);
						ii:=ii+1;
					END_WHILE
					dwSetNewPage:=awSpecialLayerGeneralActivPage[ii];
				2:	T_Visu.ptrT_ExchgParam^.T_Visu.bActivSpecialLayer:=2;
					T_Visu.ptrT_ExchgParam^.T_TouchScreenBtPanel.iStateBtLeft:=2;
					T_Visu.ptrT_ExchgParam^.T_TouchScreenNavPanel.wState:=wSpecialLayerToolRotActivTask;
					ii:=1;
					wTmp:=wSpecialLayerToolRotActivTask;
					WHILE wTmp <> 16#0 DO
						IF (wTmp AND 16#1) = 16#1 THEN EXIT; END_IF
						wTmp:=ROR(wTmp,1);
						ii:=ii+1;
					END_WHILE
					dwSetNewPage:=awSpecialLayerToolRotActivPage[ii];
				3:	T_Visu.ptrT_ExchgParam^.T_Visu.bActivSpecialLayer:=3;
					T_Visu.ptrT_ExchgParam^.T_TouchScreenBtPanel.iStateBtLeft:=4;
					T_Visu.ptrT_ExchgParam^.T_TouchScreenNavPanel.wState:=wSpecialLayerWireFeedActivTask;
					ii:=1;
					wTmp:=wSpecialLayerWireFeedActivTask;
					WHILE wTmp <> 16#0 DO
						IF (wTmp AND 16#1) = 16#1 THEN EXIT; END_IF
						wTmp:=ROR(wTmp,1);
						ii:=ii+1;
					END_WHILE
					dwSetNewPage:=awSpecialLayerWireFeedActivPage[ii];
				4:	T_Visu.ptrT_ExchgParam^.T_Visu.bActivSpecialLayer:=4;
					T_Visu.ptrT_ExchgParam^.T_TouchScreenBtPanel.iStateBtLeft:=8;
					T_Visu.ptrT_ExchgParam^.T_TouchScreenNavPanel.wState:=wSpecialLayerGrindAxisActivTask;
					ii:=1;
					wTmp:=wSpecialLayerGrindAxisActivTask;
					WHILE wTmp <> 16#0 DO
						IF (wTmp AND 16#1) = 16#1 THEN EXIT; END_IF
						wTmp:=ROR(wTmp,1);
						ii:=ii+1;
					END_WHILE
					dwSetNewPage:=awSpecialLayerGrindAxisActivPage[ii];
			ELSE
				T_Visu.ptrT_ExchgParam^.T_Visu.bActivSpecialLayer:=1;
				T_Visu.ptrT_ExchgParam^.T_TouchScreenBtPanel.iStateBtLeft:=1;
				T_Visu.ptrT_ExchgParam^.T_TouchScreenNavPanel.wState:=wSpecialLayerGeneralActivTask;
				dwSetNewPage:=wSpecialLayerGeneralActivPage;
			END_CASE;
			T_Visu.T_CtrleAction.iFunction:=6;
			T_Visu.T_CtrleAction.xExecute:=TRUE;
		END_IF;

		IF FallingEdgeSpecialLayer.Q THEN
			IF xOverlayMeasureToolDia THEN
				T_Visu.ptrT_ExchgParam^.T_FunctionCommon.xOpenOverlayMeasureInput:=FALSE;
				T_Visu.ptrT_ExchgParam^.T_FunctionCommon.xSaveButton:=FALSE;
				T_Visu.ptrT_ExchgParam^.T_FunctionCommon.xExitButton:=FALSE;
				T_Visu.ptrT_ExchgParam^.T_FunctionCommon.xHideProgressbar:=FALSE;
				xOverlayMeasureToolDia:=FALSE;
				T_Visu.T_CtrleAction.xDone:=TRUE;
			END_IF;
			IF xOverlayGrindFeedSetPlung THEN
				T_Visu.ptrT_ExchgParam^.T_FunctionCommon.xOpenOverlaySetGrindPlunge:=FALSE;
				T_Visu.ptrT_ExchgParam^.T_FunctionCommon.xSaveButton:=FALSE;
				T_Visu.ptrT_ExchgParam^.T_FunctionCommon.xExitButton:=FALSE;
				T_Visu.ptrT_ExchgParam^.T_FunctionCommon.xHideProgressbar:=FALSE;
				xOverlayGrindFeedSetPlung:=FALSE;
				T_Visu.T_CtrleAction.xDone:=TRUE;
			END_IF;
			IF T_Visu.ptrT_ExchgParam^.T_FunctionCommon.xOpenOverlayMessageBox THEN
				T_Visu.ptrT_ExchgParam^.T_FunctionCommon.xOpenOverlayMessageBox:=FALSE;
				xAction_SaveNovRAM:=FALSE;
				xAction_SaveNovRAMWithoutConfirm:=FALSE;
			END_IF;
			T_Visu.ptrT_ExchgParam^.T_Visu.bActivSpecialLayer:=0;
			T_Visu.ptrT_ExchgParam^.T_TouchScreenBtPanel.iStateBtLeft:=0;
			T_Visu.ptrT_ExchgParam^.T_TouchScreenNavPanel.wState:=wNormalLayerActivTask;
			ii:=1;
			wTmp:=wNormalLayerActivTask;
			WHILE wTmp <> 16#0 DO
				IF (wTmp AND 16#1) = 16#1 THEN EXIT; END_IF
				wTmp:=ROR(wTmp,1);
				ii:=ii+1;
			END_WHILE
			dwSetNewPage:=awNormalLayerActivPage[ii]; (*TO Do*)
			T_Visu.T_CtrleAction.iFunction:=6;
			T_Visu.T_CtrleAction.xExecute:=TRUE;
		END_IF;
		IF wActivBtLeft = 16#10 THEN
			CASE T_Visu.ptrT_ExchgParam^.T_Visu.bActivSpecialLayer OF
				1:	iTmpActivBtLeft:=1;
				2:	iTmpActivBtLeft:=2;
				3:	iTmpActivBtLeft:=4;
				4:	iTmpActivBtLeft:=8;
			END_CASE;
		ELSE
			iTmpActivBtLeft:=WORD_TO_INT(wActivBtLeft);
		END_IF;
		IF RisingEdgeBtPanelLeft.Q THEN
			iStepCounter:=iStepCounter + 1;
			CASE iTmpActivBtLeft OF
				16#1:	T_Visu.ptrT_ExchgParam^.T_Visu.bActivSpecialLayer:=1;
						T_Visu.ptrT_ExchgParam^.T_TouchScreenNavPanel.wState:=wSpecialLayerGeneralActivTask;
						dwSetNewPage:=wSpecialLayerGeneralActivPage;
				16#2:	T_Visu.ptrT_ExchgParam^.T_Visu.bActivSpecialLayer:=2;
						T_Visu.ptrT_ExchgParam^.T_TouchScreenNavPanel.wState:=wSpecialLayerToolRotActivTask;
						dwSetNewPage:=wSpecialLayerToolRotActivPage;
				16#4:	T_Visu.ptrT_ExchgParam^.T_Visu.bActivSpecialLayer:=3;
						T_Visu.ptrT_ExchgParam^.T_TouchScreenNavPanel.wState:=wSpecialLayerWireFeedActivTask;
						dwSetNewPage:=wSpecialLayerWireFeedActivPage;
				16#8:	T_Visu.ptrT_ExchgParam^.T_Visu.bActivSpecialLayer:=4;
						T_Visu.ptrT_ExchgParam^.T_TouchScreenNavPanel.wState:=wSpecialLayerGrindAxisActivTask;
						dwSetNewPage:=wSpecialLayerGrindAxisActivPage;
			END_CASE;
			bOldActivSpecialLayer:=T_Visu.ptrT_ExchgParam^.T_Visu.bActivSpecialLayer;
			IF ((wActivBtLeft AND 16#10) <> 16#10) THEN
				IF ((INT_TO_WORD(T_Visu.ptrT_ExchgParam^.T_TouchScreenBtPanel.iStateBtLeft) AND 16#10) = 16#10) THEN
					T_Visu.ptrT_ExchgParam^.T_TouchScreenBtPanel.iStateBtLeft:=WORD_TO_INT(wActivBtLeft OR 16#10);
					T_Visu.T_CtrleAction.iFunction:=3;
					T_Visu.T_CtrleAction.xExecute:=TRUE;
					xResetParaListValue:=TRUE;
				ELSE
					T_Visu.ptrT_ExchgParam^.T_TouchScreenBtPanel.iStateBtLeft:=WORD_TO_INT(wActivBtLeft);
					T_Visu.T_CtrleAction.iFunction:=6;
					T_Visu.T_CtrleAction.xExecute:=TRUE;
				END_IF;
			ELSE
				IF ((INT_TO_WORD(T_Visu.ptrT_ExchgParam^.T_TouchScreenBtPanel.iStateBtLeft) AND 16#10) = 16#10) THEN
					T_Visu.ptrT_ExchgParam^.T_TouchScreenBtPanel.iStateBtLeft:=T_Visu.ptrT_ExchgParam^.T_TouchScreenBtPanel.iStateBtLeft - 16#10;
					T_Visu.T_CtrleAction.iFunction:=6;
					T_Visu.T_CtrleAction.xExecute:=TRUE;
					xResetParaListValue:=TRUE;
				ELSE
					T_Visu.ptrT_ExchgParam^.T_TouchScreenBtPanel.iStateBtLeft:=WORD_TO_INT(wActivBtLeft OR INT_TO_WORD(T_Visu.ptrT_ExchgParam^.T_TouchScreenBtPanel.iStateBtLeft));
					T_Visu.T_CtrleAction.iFunction:=3;
					T_Visu.T_CtrleAction.xExecute:=TRUE;
					xResetParaListValue:=TRUE;
				END_IF;
			END_IF;
		END_IF;
	END_IF;
END_ACTION
ACTION CtrlPanelRightButton:
(* Management Bt Panel Right *)
	IF (T_Visu.T_PlcParam.dwActualPage = 320) THEN
		IF NOT(xMicroRodActive) THEN
		(* For MicroWire no Function for ToolFeeder-->Cancel Function F1, F2, F3 and F4 *)
			wMaskBtPanelRight:=wMaskBtPanelRight AND 16#0;
			T_Visu.ptrT_ExchgParam^.T_TouchScreenBtPanel.iNotMaskTextBt:=WORD_TO_INT(INT_TO_WORD(T_Visu.ptrT_ExchgParam^.T_TouchScreenBtPanel.iNotMaskTextBt) OR 16#3E0);
		END_IF;
	END_IF;
	IF (T_Visu.T_PlcParam.dwActualPage = 10) THEN
		IF (T_NovRam.T_Data.T_ProcessImageData.T_AutoGeometryPara.iCycleGeometry <= 1) THEN
			T_Visu.ptrT_ExchgParam^.T_TouchScreenBtPanel.iNotMaskTextBt:=WORD_TO_INT(INT_TO_WORD(T_Visu.ptrT_ExchgParam^.T_TouchScreenBtPanel.iNotMaskTextBt) OR 16#1E0);
		END_IF;
	END_IF;
	TimerPressBtPanelRight(IN:=TRUE, PT:=T#3600s);
	IF T_Visu.ptrT_ExchgParam^.T_Config.xNoTouchScreenBtPanel THEN
		wActivBtRight:=wSPSSpecialButton;
	ELSE
		wActivBtRight:=INT_TO_WORD(T_Visu.ptrT_ExchgParam^.T_TouchScreenBtPanel.iActivBtRight);
	END_IF;
	RisingEdgeBtPanelRight(CLK:=(wActivBtRight AND wMaskBtPanelRight) <> 16#0);
	FallingEdgeBtPanelRight(CLK:=(wActivBtRight AND wMaskBtPanelRight) <> 16#0);
	xTmp:=	(NOT(xChangePage)
			AND T_Visu.T_CtrleAction.xDone
			AND NOT(T_Visu.T_CtrleAction.xExecute)
			AND NOT(T_StartUp.T_State.xBlockChangeMovementVisu)
			(*AND NOT(T_StartUp.T_State.xBlockVisuNavigation)*))
			OR xDelayActionBtPanelRight;
	IF (wActivBtRight = 0) AND NOT(xDelayActionBtPanelRight) THEN
		TimerPressBtPanelRight(IN:=FALSE);
	END_IF;
	IF xTmp THEN
		(* Rising edge action *)
		IF RisingEdgeBtPanelRight.Q AND (bButtonPanelLocked = 16#0) AND (NOT(T_StartUp.T_State.xBlockVisuNavigation)
		OR ((T_NovRam.T_Data.T_ProcessImageData.T_AutoGeometryPara.iCycleGeometry > 1)) AND (T_Visu.T_PlcParam.dwActualPage = 10)) THEN
		(* init. variable *)
			ii:=1;
			wTmp:=wActivBtRight;
			wTmpActivBtRight:=wActivBtRight;
			wTmp:=ROR(wTmp,5);
			(* only one button is used *)
			WHILE wTmp <> 16#0 DO
				IF (wTmp AND 16#1) = 16#1 THEN EXIT; END_IF
				wTmp:=ROR(wTmp,1);
				ii:=ii+1;
			END_WHILE
		(* SOA 09.12.2022 { *)
			(* set the new action if present *)
			IF (T_Visu.T_PlcParam.dwActualPage = 120) OR (T_Visu.T_PlcParam.dwActualPage = 121) OR (T_Visu.T_PlcParam.dwActualPage = 140) OR (T_Visu.T_PlcParam.dwActualPage = 141) THEN
				dwSetNewPage := ( T_ConfigPage.aiRTrigActionPanelRight[ii] - 10000);
				T_Visu.T_CtrleAction.iFunction:=7;
				T_Visu.T_CtrleAction.xExecute:=TRUE;
			ELSIF T_ConfigPage.aiRTrigActionPanelRight[ii] <> 0 THEN
				T_Visu.T_CtrleAction.iFunction:=T_ConfigPage.aiRTrigActionPanelRight[ii];
				T_Visu.T_CtrleAction.xExecute:=TRUE;
			END_IF
		(* SOA 09.12.2022  } *)
			IF (T_ConfigPage.aiFTrigActionPanelRight[ii] = 301) THEN
				xTmpStopAxis:=TRUE;
			END_IF
			(* init. timer press button *)
			TimerPressBtPanelRight(IN:=FALSE);
			(* Lock button panel *)
			bButtonPanelLocked:=16#2;
			(* init. variable *)
			xDelayActionBtPanelRight:=FALSE;
		END_IF
		(* Falling Edge action activ only if the delay action has been started *)
		IF FallingEdgeBtPanelRight.Q AND ((bButtonPanelLocked AND 16#2) = 16#2) THEN
			ii:=1;
			wTmp:=wTmpActivBtRight;
			wTmp:=ROR(wTmp,5);
			(* only one button is used *)
			WHILE wTmp <> 16#0 DO
				IF (wTmp AND 16#1) = 16#1 THEN EXIT; END_IF
				wTmp:=ROR(wTmp,1);
				ii:=ii+1;
			END_WHILE
			(* set the new action if present *)
			IF T_ConfigPage.aiFTrigActionPanelRight[ii] <> 0 (*AND xDelayActionBtPanelRight*) THEN
				T_Visu.T_CtrleAction.iFunction:=T_ConfigPage.aiFTrigActionPanelRight[ii];
				T_Visu.T_CtrleAction.xExecute:=TRUE;
				IF (T_Visu.T_CtrleAction.iFunction = 301) THEN
					xTmpStopAxis:=TRUE;
				END_IF;
			END_IF
			(* release lock panel *)
			bButtonPanelLocked:=bButtonPanelLocked XOR 16#2;
			(* init. variable *)
			xDelayActionBtPanelRight:=FALSE;
		END_IF;

		(* monitor delay *)
		xTmp:=	NOT(xDelayActionBtPanelRight)
				AND NOT(FallingEdgeBtPanelRight.Q)
				AND (bButtonPanelLocked AND 16#2) =16#2;
		IF xTmp AND (TimerPressBtPanelRight.ET > T#500ms) THEN
		(* activ delay action *)
			ii:=1;
			wTmp:=wActivBtRight;
			wTmp:=ROR(wTmp,5);
			(* only one button is used *)
			WHILE wTmp <> 16#0 DO
				IF (wTmp AND 16#1) = 16#1 THEN EXIT; END_IF
				wTmp:=ROR(wTmp,1);
				ii:=ii+1;
			END_WHILE
			(* set the new action if present *)
			IF T_ConfigPage.aiDelayActionPanelRight[ii] <> 0 THEN
				T_Visu.T_CtrleAction.iFunction:=T_ConfigPage.aiDelayActionPanelRight[ii];
				T_Visu.T_CtrleAction.xExecute:=TRUE;
			END_IF
			(* confirm execution delay action *)
			xDelayActionBtPanelRight:=TRUE;
		END_IF;
		IF T_Visu.T_CtrleAction.xDone AND (wActivBtRight = 16#0) AND (bButtonPanelLocked = 16#2) THEN
			bButtonPanelLocked:=0;
		END_IF;
	END_IF
	IF xTmpStopAxis THEN
		IF ptrTeachINAxis^.T_CtrleSingle.xErr THEN
			IF (ptrTeachINAxis^.T_Config_Gen.iTyp <> 0) THEN
				diErrorNr:=(ptrTeachINAxis^.T_Config_Gen.iTyp * 1000000) + ptrTeachINAxis^.T_CtrleSingle.udiErrorID;
			ELSE
				diErrorNr:=0;
			END_IF;
			FBErrorMessage(	diErrorNr:=diErrorNr,
							T_ErrorList:=T_ErrorList);
			T_Visu.ptrT_ExchgParam^.T_Visu.T_Message.sDynamicTextEnglish:=FBErrorMessage.sErrorTextEnglish;
			T_Visu.ptrT_ExchgParam^.T_Visu.T_Message.sDynamicTextDeutsch:=FBErrorMessage.sErrorTextDeutsch;
			T_Visu.ptrT_ExchgParam^.T_Visu.T_Message.sDynamicTextFrancais:=FBErrorMessage.sErrorTextFrancais;
			T_Visu.ptrT_ExchgParam^.T_SafetyCtrl.xSetForceError:=TRUE;
			T_Visu.ptrT_ExchgParam^.T_SafetyCtrl.diSetForceErrorNr:=diErrorNr;
			ptrTeachINAxis^.T_CtrleSingle.iFunction:=1;
			ptrTeachINAxis^.T_CtrleSingle.xExecute:=TRUE;
			T_StartUp.T_Ctrle.xSetSecurityStateON:=TRUE;
		END_IF;
	END_IF;
	IF xTmpStopAxis AND T_Visu.T_CtrleAction.xDone AND (bButtonPanelLocked = 0) AND NOT(T_Visu.T_CtrleAction.xExecute) AND (NOT(T_Station.THardware.TAxisToolLeft.T_CtrleSingle.xNotMoving) OR
	    (NOT(T_Station.THardware.TAxisToolCenter.T_CtrleSingle.xNotMoving) AND xMicroRodActive) OR NOT(T_Station.THardware.TAxisToolRight.T_CtrleSingle.xNotMoving) OR
	     NOT(T_Station.THardware.TAxisToolFeeder.T_CtrleSingle.xNotMoving) OR NOT(T_Station.THardware.TAxisGrindFeeder.T_CtrleSingle.xNotMoving)) THEN
		T_Visu.T_CtrleAction.iFunction:=301;
		T_Visu.T_CtrleAction.xExecute:=TRUE;
	END_IF;
	IF xTmpStopAxis AND T_Visu.T_CtrleAction.xDone AND NOT(T_Visu.T_CtrleAction.xExecute) AND T_Station.THardware.TAxisToolLeft.T_CtrleSingle.xNotMoving AND
	    ((T_Station.THardware.TAxisToolCenter.T_CtrleSingle.xNotMoving AND xMicroRodActive) OR NOT(xMicroRodActive)) AND T_Station.THardware.TAxisToolRight.T_CtrleSingle.xNotMoving AND
	    T_Station.THardware.TAxisToolFeeder.T_CtrleSingle.xNotMoving AND T_Station.THardware.TAxisGrindFeeder.T_CtrleSingle.xNotMoving THEN
		xTmpStopAxis:=FALSE;
	END_IF;
END_ACTION
ACTION CtrlProcessFunction:
(* Manage process execution *)
	(* ...done *)
	RisingEdgeProcessDone(CLK:=T_Visu.T_CtrleProcess.xDone);
	IF RisingEdgeProcessDone.Q THEN
		IF NOT(T_StartUp.T_State.xBlockChangeMovementVisu) THEN
			IF T_Visu.T_CtrleProcess.iFunction <> 0 AND T_Visu.ptrT_ExchgParam^.T_Visu.T_Message.iState = 0 THEN
			(* call confirmation message *)
				IF NOT xStopImmediatly THEN
					IF (T_Visu.T_PlcParam.dwActualPage = 110) THEN
						T_Visu.ptrT_ExchgParam^.T_Visu.T_Message.iState:=22;
					END_IF;
					(*T_Visu.ptrT_ExchgParam^.T_Visu.T_Message.iState
						:=iFctReturnConfMessage(iNumAction:=T_Process.iFunctNr+1100);*);
				(* Display message 'Process is aborded' *)
				ELSE T_Visu.ptrT_ExchgParam^.T_Visu.T_Message.iState:=9; END_IF
			END_IF
		END_IF;
	END_IF
	(* ...error *)
	RisingEdgeProcessError(CLK:=T_Visu.T_CtrleProcess.xErr);
	IF RisingEdgeProcessError.Q THEN
	(* call function bloc action error *)
		IF NOT(T_StartUp.T_State.xBlockChangeMovementVisu) THEN
			(*
			fbQvisError(	udiActionError:=T_Visu.T_CtrleProcess.udiErrorID,
						T_Message:=T_Visu.ptrT_ExchgParam^.T_Visu.T_Message);
			*);
		END_IF;
		(* Init. variable *)
		T_Visu.T_CtrleProcess.xExecute:=FALSE;
		T_Visu.T_CtrleProcess.xDone:=TRUE;
		T_Visu.T_CtrleProcess.xErr:=FALSE;
		T_Visu.T_CtrleProcess.udiErrorID:=0;
		(*iStepProcess:=1;*)
		(*xStepProcessDone:=FALSE;*)
	END_IF
	(* ...reset *)
	RisingEdgeResetProcess(CLK:=T_Visu.T_CtrleProcess.xReset);
	IF RisingEdgeResetProcess.Q THEN
		(* Init. variable *)
		T_Visu.T_CtrleProcess.xExecute:=FALSE;
		T_Visu.T_CtrleProcess.xDone:=TRUE;
		T_Visu.T_CtrleProcess.xErr:=FALSE;
		T_Visu.T_CtrleProcess.udiErrorID:=0;
		(*iStepProcess:=1;*)
		(*xStepProcessDone:=FALSE;*)
		(* Release process *)
		T_Visu.T_CtrleProcess.xReset:=FALSE;
	END_IF
	RisingEdgeExecuteProcess(CLK:=T_Visu.T_CtrleProcess.xExecute);
	IF RisingEdgeExecuteProcess.Q THEN
		(* Release execution *)
		T_Visu.T_CtrleProcess.xExecute:=FALSE;
		CASE T_Visu.T_CtrleProcess.iFunction OF
		(* Process machine *)
		1:	xProcessMachine:=TRUE;
		(* Process station *)
		2:	xProcessStation:=TRUE;
		(* process not implemented *)
		ELSE	T_Visu.T_CtrleProcess.xDone:=FALSE;
				T_Visu.T_CtrleProcess.xErr:=TRUE;
				T_Visu.T_CtrleProcess.udiErrorID:=16#E000;
				(* exit FB *)
				RETURN;
		END_CASE
		(* Init. variable *)
		T_Visu.T_CtrleProcess.xDone:=FALSE;
		T_Visu.T_CtrleProcess.xErr:=FALSE;
		T_Visu.T_CtrleProcess.udiErrorID:=0;
		iStepProcess:=1;
		xStepProcessDone:=FALSE;
		(* exit FB *)
		RETURN;
	END_IF

(* Process machine *)
	IF xProcessMachine OR xProcessStation THEN
		CASE iStepProcess OF
	(* SOA 22.02.2023  {  *)
		1: 	IF  (T_Visu.T_PlcParam.dwActualPage = 10) AND T_ExchgParam.T_StationCommon.T_AutoGeometryPara.xWarmUp THEN
					iStepProcess:=2;
				ELSE
					iStepProcess:=4;
			END_IF
		2:	(* Overlay Message Error *)
			T_VisuQVis.ptrT_ExchgParam^.T_SafetyCtrl.bStateMessageError:=0;
			T_VisuQVis.ptrT_ExchgParam^.T_SafetyCtrl.bStateMessageInfo:=0;
			T_VisuQVis.ptrT_ExchgParam^.T_SafetyCtrl.bStateMessageWarning:=1;
			T_VisuQVis.ptrT_ExchgParam^.T_SafetyCtrl.iMsgInfoLine1:=6;	(* BOOTING OF THE MACHINE COMPLEATED! *)
			T_VisuQVis.ptrT_ExchgParam^.T_SafetyCtrl.iMsgInfoLine2:=6;	(* CONFIRM AND THE MACHINE *)
			T_VisuQVis.ptrT_ExchgParam^.T_SafetyCtrl.iMsgInfoLine3:=6;	(* WILL BE READY TO USE IT! *)
			T_VisuQVis.ptrT_ExchgParam^.T_SafetyCtrl.iMsgInfoLine4:=6;	(*  *)
			T_VisuQVis.ptrT_ExchgParam^.T_SafetyCtrl.xConfirmMsgWarning:=FALSE;
			T_VisuQVis.ptrT_ExchgParam^.T_SafetyCtrl.xBlockVisuObject:=TRUE;
			(*xRdy:=TRUE; *)
			(* next step *)
			iStepProcess:=3;
		3:	IF T_VisuQVis.ptrT_ExchgParam^.T_SafetyCtrl.xConfirmMsgWarning THEN
				T_VisuQVis.ptrT_ExchgParam^.T_SafetyCtrl.xBlockVisuObject:=FALSE;
				T_VisuQVis.ptrT_ExchgParam^.T_SafetyCtrl.bStateMessageWarning:=0;
				T_VisuQVis.ptrT_ExchgParam^.T_SafetyCtrl.xConfirmMsgWarning:=FALSE;
				T_VisuQVis.ptrT_ExchgParam^.T_SafetyCtrl.bStateAutoGeometry:=1;
				T_VisuQVis.ptrT_ExchgParam^.T_SafetyCtrl.bStateAutoGroove:=1;
				T_VisuQVis.ptrT_ExchgParam^.T_SafetyCtrl.bStateReference:=1;
				T_VisuQVis.ptrT_ExchgParam^.T_SafetyCtrl.bStateToolCalibration:=1;
				T_VisuQVis.ptrT_ExchgParam^.T_SafetyCtrl.bStateToolTorque:=1;
				T_VisuQVis.ptrT_ExchgParam^.T_SafetyCtrl.bStateTeachInToolLeft:=1;
				T_VisuQVis.ptrT_ExchgParam^.T_SafetyCtrl.bStateTeachInToolCenter:=1;
				T_VisuQVis.ptrT_ExchgParam^.T_SafetyCtrl.bStateTeachInToolRight:=1;
				T_VisuQVis.ptrT_ExchgParam^.T_SafetyCtrl.bStateTeachInToolFeeder:=1;
				T_VisuQVis.ptrT_ExchgParam^.T_SafetyCtrl.bStateTeachInGrindFeeder:=1;
				T_VisuQVis.ptrT_ExchgParam^.T_StationCommon.iWireFeederRefIndexState:=1;
				(* next step *)
				iStepProcess:=4;
			END_IF
	(* SOA 22.02.2023  }  *)
		4:	(* next step *)
			T_Process.xStart:=TRUE;
			iStepProcess:=10;
			IF (T_Visu.T_PlcParam.dwActualPage = 10) THEN
				T_Visu.ptrT_ExchgParam^.T_SafetyCtrl.bStateAutoGeometry:=2;
			ELSIF (T_Visu.T_PlcParam.dwActualPage = 20) THEN
				T_Visu.ptrT_ExchgParam^.T_SafetyCtrl.bStateAutoGroove:=2;
			ELSIF (T_Visu.T_PlcParam.dwActualPage = 30) THEN
				T_Visu.ptrT_ExchgParam^.T_SafetyCtrl.bStateReference:=2;
			ELSIF (T_Visu.T_PlcParam.dwActualPage = 110) THEN
				T_Visu.ptrT_ExchgParam^.T_SafetyCtrl.bStateToolCalibration:=2;
			END_IF;
			xStepProcessDone:=FALSE;
		(* wait confirmation *)
		10:	IF NOT(xStepProcessDone) THEN
			(* release execution *)
				T_Process.xStart:=FALSE;
				xStepProcessDone:=TRUE;
				IF T_Visu.ptrT_ExchgParam^.T_StationCommon.T_AutoGeometryPara.xWarmUp THEN
					xWarmUpMessageActiv:=TRUE;
					xWarmUpMessageDone:=TRUE;
				END_IF;
			ELSE
				IF T_Process.xEnd THEN
					(* action done *)
					iStepProcess:=90;
					xStepProcessDone:=FALSE;
				ELSE
					IF T_Visu.ptrT_ExchgParam^.T_StationCommon.T_AutoGeometryPara.xWarmUp AND xWarmUpMessageActiv THEN
						T_Visu.ptrT_ExchgParam^.T_Visu.T_Message.iState:=124;	(* WarmUp cycle activ *)
						xWarmUpMessageActiv:=FALSE;
					END_IF;
					IF (T_Visu.ptrT_ExchgParam^.T_Visu.T_Message.iState=124                                                 )	AND
					     NOT(T_Visu.ptrT_ExchgParam^.T_StationCommon.T_AutoGeometryPara.xWarmUp) 	AND
					     xWarmUpMessageDone 															THEN
						T_Visu.ptrT_ExchgParam^.T_Visu.T_Message.iState:=125;	(*WarmUp cycle time arrived. <Press StopButton>*)
						xWarmUpMessageDone:=FALSE;
					END_IF;
					IF T_Process.xError THEN
						(* action error *)
						iStepProcess:=99;
						xStepProcessDone:=FALSE;
						IF xProcessMachine THEN
							T_Visu.ptrT_ExchgParam^.T_TouchScreenBtPanel.iStateBtLeft:=0;
							IF(T_Process.iFunctNr = 10) THEN
								IF (T_Visu.T_PlcParam.dwActualPage <> 10) THEN
									T_Visu.T_PlcParam.dwSetNewPage:=10;
									T_Visu.T_CtrleVisu.iFunction:=1;
									T_Visu.T_CtrleVisu.xExecute:=TRUE;
								END_IF;
							END_IF;
							IF(T_Process.iFunctNr = 20) THEN
								IF (T_Visu.T_PlcParam.dwActualPage <> 20) THEN
									T_Visu.T_PlcParam.dwSetNewPage:=20;
									T_Visu.T_CtrleVisu.iFunction:=1;
									T_Visu.T_CtrleVisu.xExecute:=TRUE;
								END_IF;
							END_IF;
							IF(T_Process.iFunctNr = 30) THEN
								IF (T_Visu.T_PlcParam.dwActualPage <> 30) THEN
									T_Visu.T_PlcParam.dwSetNewPage:=30;
									T_Visu.T_CtrleVisu.iFunction:=1;
									T_Visu.T_CtrleVisu.xExecute:=TRUE;
								END_IF;
							END_IF;
							IF(T_Process.iFunctNr = 40) THEN
								IF (T_Visu.T_PlcParam.dwActualPage <> 110) THEN
									T_Visu.T_PlcParam.dwSetNewPage:=110;
									T_Visu.T_CtrleVisu.iFunction:=1;
									T_Visu.T_CtrleVisu.xExecute:=TRUE;
								END_IF;
							END_IF;
						END_IF;
					END_IF
				END_IF
				IF NOT(T_TwinSafeOut.QxContactor_K3) OR NOT(T_TwinSafeOut.QxContactor_K4) THEN
					(*T_Process.xEnable:=FALSE;*)
					(*iStepProcess:=21;*)
					iStepProcess:=99;
					RETURN;
				END_IF;
			END_IF
		21:	IF NOT(T_Process.xEnd) THEN
				T_Process.xEnable:=TRUE;
				iStepProcess:=22;
			ELSE
				T_Process.xEnable:=FALSE;
			END_IF;
		22:	IF T_Process.xEnd THEN
				T_Visu.T_CtrleProcess.xDone:=TRUE;
				T_Visu.T_CtrleProcess.xErr:=FALSE;
				T_Visu.T_CtrleProcess.udiErrorID:=0;
				xProcessMachine:=FALSE;
				xProcessStation:=FALSE;
			END_IF;
		(* call page *)
		30:	T_Visu.T_PlcParam.dwSetNewPage:=dwPageNrProcessStart;
			T_Visu.T_CtrleVisu.iFunction:=2;
			T_Visu.T_CtrleVisu.xExecute:=TRUE;
			(* next step *)
			iStepProcess:=90;
		(* process done *)
		90:	IF NOT(T_Visu.T_CtrleVisu.xExecute) AND T_Visu.T_CtrleVisu.xDone THEN
				T_StartUp.T_State.xBlockChangeMovementVisu:=FALSE;
				IF (T_Visu.T_PlcParam.dwActualPage = 10) THEN
					T_Visu.ptrT_ExchgParam^.T_SafetyCtrl.bStateAutoGeometry:=1;
				ELSIF (T_Visu.T_PlcParam.dwActualPage = 20) THEN
					T_Visu.ptrT_ExchgParam^.T_SafetyCtrl.bStateAutoGroove:=1;
				ELSIF (T_Visu.T_PlcParam.dwActualPage = 30) THEN
					T_Visu.ptrT_ExchgParam^.T_SafetyCtrl.bStateReference:=1;
				ELSIF (T_Visu.T_PlcParam.dwActualPage = 110) THEN
					T_Visu.ptrT_ExchgParam^.T_SafetyCtrl.bStateToolCalibration:=1;
				END_IF;
				IF xProcessMachine THEN
					IF NOT(T_StartUp.T_State.xBlockChangeMovementVisu) THEN
						T_StartUp.T_Ctrle.xExecute:=TRUE;
						T_StartUp.T_Ctrle.iFunction:=11;	(* Acitvate Info Message Overlay *)
						IF (T_Process.iFunctNr = 30) THEN
							(* THE REFERENCE DRIVE  IS COMPLEATED! *)
							(* CONFIRM THIS MESSAGE AND *)
							(* THE MACHINE WILL BE READY! *)
							(*  *)
							T_StartUp.T_Ctrle.iMsgNumber:=3;
						END_IF;
						IF (T_Process.iFunctNr = 10) OR (T_Process.iFunctNr = 20) THEN
							(* THE  AUTO MODE CYCLE IS COMPLEATED! *)
							(* CONFIRM THIS MESSAGE AND *)
							(* THE MACHINE WILL BE READY! *)
							(*  *)
							T_StartUp.T_Ctrle.iMsgNumber:=2;
						END_IF;
					END_IF;
				END_IF;
				T_Visu.T_CtrleProcess.xDone:=TRUE;
				T_Visu.T_CtrleProcess.xErr:=FALSE;
				T_Visu.T_CtrleProcess.udiErrorID:=0;
				xProcessMachine:=FALSE;
				xProcessStation:=FALSE;
			END_IF;
		(* error *)
		99:	IF NOT(T_Visu.T_CtrleVisu.xExecute) AND T_Visu.T_CtrleVisu.xDone THEN
				T_StartUp.T_State.xBlockChangeMovementVisu:=FALSE;
				IF xProcessMachine THEN
					T_StartUp.T_Ctrle.xExecute:=TRUE;
					T_StartUp.T_Ctrle.iFunction:=10;	(* Activate Error Message Overlay *)
					IF (T_Process.iFunctNr = 30) THEN
						(* DURING MACHINE REFERENCE PROC. *)
						(* AN ERROR HAS OCCURRED *)
						(* PLEASE CONFIRM  AND CHECK *)
						(* THE ACCORDING ERROR *)
						T_StartUp.T_Ctrle.iMsgNumber:=14;
					END_IF;
					IF (T_Process.iFunctNr = 10) OR (T_Process.iFunctNr = 20) THEN
						(* DURING THE AUTO MODE *)
						(* AN ERROR HAS OCCURRED *)
						(* PLEASE CONFIRM AND CHECK *)
						(* THE ACCORDING ERROR *)
						T_StartUp.T_Ctrle.iMsgNumber:=13;
					END_IF;
				END_IF;
				T_Visu.T_CtrleProcess.xDone:=FALSE;
				T_Visu.T_CtrleProcess.xErr:=TRUE;
				T_Visu.T_CtrleProcess.udiErrorID:=16#E0000 + T_Visu.T_CtrleProcess.iFunction;
				xProcessMachine:=FALSE;
				xProcessStation:=FALSE;
			END_IF;
		END_CASE
	END_IF
END_ACTION
ACTION CtrlStartStopButton:
(************************************************************************************************************************************************************************)
(********start of the managment of the external start-stop button, special button and function button and task button and external tool buttons********)
(************************************************************************************************************************************************************************)
(* Start button *)
	(* ...manage action button *)
	xTmp:=	NOT(xChangePage)
			AND (T_Visu.T_CtrleAction.xDone)
			AND NOT(T_Visu.T_CtrleAction.xExecute);
	IF xTmp THEN
		(* manage rising edge start button *)
		RisingEdgeStartButton(CLK:=xStartButton AND T_ConfigPage.xMaskBtStart);
		IF RisingEdgeStartButton.Q AND bButtonPanelLocked = 16#0 AND NOT(T_StartUp.T_State.xBlockChangeMovementVisu) THEN
		(* panel locked *)
			bButtonPanelLocked:=16#10;
			(* Start process at the begin *)
			T_Visu.T_CtrleAction.xExecute:=TRUE;
			CASE T_Visu.T_PlcParam.dwActualPage OF
			(* Data machine *)
			10:	T_Visu.T_CtrleAction.iFunction:=710;
			20:	T_Visu.T_CtrleAction.iFunction:=720;
			30:	T_Visu.T_CtrleAction.iFunction:=730;
			110:	T_Visu.T_CtrleAction.iFunction:=640;
			210:	T_Visu.T_CtrleAction.iFunction:=318;
			220:	T_Visu.T_CtrleAction.iFunction:=402;
			310:	T_Visu.T_CtrleAction.iFunction:=305;
			330:	T_Visu.T_CtrleAction.iFunction:=420;
			410:	CASE T_Visu.ptrT_ExchgParam^.T_TeachIn.iSelectAxisGrind OF
				1:	T_Visu.T_CtrleAction.iFunction:=305;
				2:	T_Visu.T_CtrleAction.iFunction:=318;
				END_CASE
			ELSE
				T_Visu.T_CtrleAction.xExecute:=FALSE;
			END_CASE
			(* save page number for stop procedure *)
			IF T_Visu.T_CtrleAction.xExecute THEN
				dwPageNrProcessStart:=T_Visu.T_PlcParam.dwActualPage;
				xStopImmediatly:=FALSE;
			END_IF
		END_IF
		(* manage falling edge start button *)
		FallingEdgeStartButton(CLK:=xStartButton AND T_ConfigPage.xMaskBtStart);
		IF FallingEdgeStartButton.Q AND (bButtonPanelLocked AND 16#10) = 16#10 THEN bButtonPanelLocked:=bButtonPanelLocked XOR 16#10; END_IF
	ELSE
		RisingEdgeStartButton(CLK:=FALSE);
		FallingEdgeStartButton(CLK:=TRUE);
	END_IF

